# B&R Automation Studio project NAINV104C00R8L515F00 (part 7)

#### fHermesFormBoardArrived.st
```iecst
(* Hermes Form Board Arrived Table Data (Total Index Written In Table) *)
FUNCTION fHermesFormBoardArrived

	memset(ADR(pa_tyXMLTable) , 0 , SIZEOF(pa_tyXMLTable));
	iTotalIdxWrite	:= 0;

	fHermesGetTimestamp(ADR(sTimestamp) , tyDTStructure);

	pa_tyXMLTable[iTotalIdxWrite].sTitle	:= 'ST';
	pa_tyXMLTable[iTotalIdxWrite].sValue	:= 'Hermes';
	pa_tyXMLTable[iTotalIdxWrite].uiSize	:= LEN(pa_tyXMLTable[iTotalIdxWrite].sValue);

	iTotalIdxWrite	:= iTotalIdxWrite + 1;

	pa_tyXMLTable[iTotalIdxWrite].sTitle	:= 'AT';
	pa_tyXMLTable[iTotalIdxWrite].sValue	:= 'Timestamp';
	pa_tyXMLTable[iTotalIdxWrite].uiSize	:= LEN(pa_tyXMLTable[iTotalIdxWrite].sValue);

	iTotalIdxWrite	:= iTotalIdxWrite + 1;

	pa_tyXMLTable[iTotalIdxWrite].sTitle	:= 'AV';
	pa_tyXMLTable[iTotalIdxWrite].sValue	:= sTimestamp;
	pa_tyXMLTable[iTotalIdxWrite].uiSize	:= LEN(pa_tyXMLTable[iTotalIdxWrite].sValue);

	iTotalIdxWrite	:= iTotalIdxWrite + 1;

	pa_tyXMLTable[iTotalIdxWrite].sTitle	:= 'EN';
	pa_tyXMLTable[iTotalIdxWrite].sValue	:= '';
	pa_tyXMLTable[iTotalIdxWrite].uiSize	:= LEN(pa_tyXMLTable[iTotalIdxWrite].sValue);

	iTotalIdxWrite	:= iTotalIdxWrite + 1;

	pa_tyXMLTable[iTotalIdxWrite].sTitle	:= 'ST';
	pa_tyXMLTable[iTotalIdxWrite].sValue	:= 'BoardArrived';
	pa_tyXMLTable[iTotalIdxWrite].uiSize	:= LEN(pa_tyXMLTable[iTotalIdxWrite].sValue);

	iTotalIdxWrite	:= iTotalIdxWrite + 1;

	IF tyParameter.tyAvl.bMachineId = TRUE THEN
		pa_tyXMLTable[iTotalIdxWrite].sTitle	:= 'AT';
		pa_tyXMLTable[iTotalIdxWrite].sValue	:= 'MachineId';
		pa_tyXMLTable[iTotalIdxWrite].uiSize	:= LEN(pa_tyXMLTable[iTotalIdxWrite].sValue);

		iTotalIdxWrite	:= iTotalIdxWrite + 1;

		pa_tyXMLTable[iTotalIdxWrite].sTitle	:= 'AV';
		pa_tyXMLTable[iTotalIdxWrite].sValue	:= tyParameter.tyData.sMachineId;
		pa_tyXMLTable[iTotalIdxWrite].uiSize	:= LEN(pa_tyXMLTable[iTotalIdxWrite].sValue);

		iTotalIdxWrite	:= iTotalIdxWrite + 1;
	END_IF

	IF tyParameter.tyAvl.bUpstreamLaneId = TRUE THEN
		pa_tyXMLTable[iTotalIdxWrite].sTitle	:= 'AT';
		pa_tyXMLTable[iTotalIdxWrite].sValue	:= 'UpstreamLaneId';
		pa_tyXMLTable[iTotalIdxWrite].uiSize	:= LEN(pa_tyXMLTable[iTotalIdxWrite].sValue);

		iTotalIdxWrite	:= iTotalIdxWrite + 1;

		pa_tyXMLTable[iTotalIdxWrite].sTitle	:= 'AV';
		pa_tyXMLTable[iTotalIdxWrite].sValue	:= UDINT_TO_STRING(tyParameter.tyData.iUpstreamLaneId);
		pa_tyXMLTable[iTotalIdxWrite].uiSize	:= LEN(pa_tyXMLTable[iTotalIdxWrite].sValue);

		iTotalIdxWrite	:= iTotalIdxWrite + 1;
	END_IF

	IF tyParameter.tyAvl.bUpstreamInterfaceId = TRUE THEN
		pa_tyXMLTable[iTotalIdxWrite].sTitle	:= 'AT';
		pa_tyXMLTable[iTotalIdxWrite].sValue	:= 'UpstreamInterfaceId';
		pa_tyXMLTable[iTotalIdxWrite].uiSize	:= LEN(pa_tyXMLTable[iTotalIdxWrite].sValue);

		iTotalIdxWrite	:= iTotalIdxWrite + 1;

		pa_tyXMLTable[iTotalIdxWrite].sTitle	:= 'AV';
		pa_tyXMLTable[iTotalIdxWrite].sValue	:= tyParameter.tyData.sUpstreamInterfaceId;
		pa_tyXMLTable[iTotalIdxWrite].uiSize	:= LEN(pa_tyXMLTable[iTotalIdxWrite].sValue);

		iTotalIdxWrite	:= iTotalIdxWrite + 1;
	END_IF

	IF tyParameter.tyAvl.bMagazineId = TRUE THEN
		pa_tyXMLTable[iTotalIdxWrite].sTitle	:= 'AT';
		pa_tyXMLTable[iTotalIdxWrite].sValue	:= 'MagazineId';
		pa_tyXMLTable[iTotalIdxWrite].uiSize	:= LEN(pa_tyXMLTable[iTotalIdxWrite].sValue);

		iTotalIdxWrite	:= iTotalIdxWrite + 1;

		pa_tyXMLTable[iTotalIdxWrite].sTitle	:= 'AV';
		pa_tyXMLTable[iTotalIdxWrite].sValue	:= tyParameter.tyData.sMagazineId;
		pa_tyXMLTable[iTotalIdxWrite].uiSize	:= LEN(pa_tyXMLTable[iTotalIdxWrite].sValue);

		iTotalIdxWrite	:= iTotalIdxWrite + 1;
	END_IF

	IF tyParameter.tyAvl.bSlotId = TRUE THEN
		pa_tyXMLTable[iTotalIdxWrite].sTitle	:= 'AT';
		pa_tyXMLTable[iTotalIdxWrite].sValue	:= 'SlotId';
		pa_tyXMLTable[iTotalIdxWrite].uiSize	:= LEN(pa_tyXMLTable[iTotalIdxWrite].sValue);

		iTotalIdxWrite	:= iTotalIdxWrite + 1;

		pa_tyXMLTable[iTotalIdxWrite].sTitle	:= 'AV';
		pa_tyXMLTable[iTotalIdxWrite].sValue	:= UDINT_TO_STRING(tyParameter.tyData.iSlotId);
		pa_tyXMLTable[iTotalIdxWrite].uiSize	:= LEN(pa_tyXMLTable[iTotalIdxWrite].sValue);

		iTotalIdxWrite	:= iTotalIdxWrite + 1;
	END_IF

	IF tyParameter.tyAvl.bBoardTransfer = TRUE THEN
		pa_tyXMLTable[iTotalIdxWrite].sTitle	:= 'AT';
		pa_tyXMLTable[iTotalIdxWrite].sValue	:= 'BoardTransfer';
		pa_tyXMLTable[iTotalIdxWrite].uiSize	:= LEN(pa_tyXMLTable[iTotalIdxWrite].sValue);

		iTotalIdxWrite	:= iTotalIdxWrite + 1;

		pa_tyXMLTable[iTotalIdxWrite].sTitle	:= 'AV';
		pa_tyXMLTable[iTotalIdxWrite].sValue	:= DINT_TO_STRING(UDINT_TO_DINT(tyParameter.tyData.eBoadTransfer));
		pa_tyXMLTable[iTotalIdxWrite].uiSize	:= LEN(pa_tyXMLTable[iTotalIdxWrite].sValue);

		iTotalIdxWrite	:= iTotalIdxWrite + 1;
	END_IF

	IF tyParameter.tyAvl.bBoardId = TRUE THEN
		pa_tyXMLTable[iTotalIdxWrite].sTitle	:= 'AT';
		pa_tyXMLTable[iTotalIdxWrite].sValue	:= 'BoardId';
		pa_tyXMLTable[iTotalIdxWrite].uiSize	:= LEN(pa_tyXMLTable[iTotalIdxWrite].sValue);

		iTotalIdxWrite	:= iTotalIdxWrite + 1;

		pa_tyXMLTable[iTotalIdxWrite].sTitle	:= 'AV';
		pa_tyXMLTable[iTotalIdxWrite].sValue	:= tyParameter.tyData.sBoardId;
		pa_tyXMLTable[iTotalIdxWrite].uiSize	:= LEN(pa_tyXMLTable[iTotalIdxWrite].sValue);

		iTotalIdxWrite	:= iTotalIdxWrite + 1;
	END_IF

	IF tyParameter.tyAvl.bBoardIdCreatedBy = TRUE THEN
		pa_tyXMLTable[iTotalIdxWrite].sTitle	:= 'AT';
		pa_tyXMLTable[iTotalIdxWrite].sValue	:= 'BoardIdCreatedBy';
		pa_tyXMLTable[iTotalIdxWrite].uiSize	:= LEN(pa_tyXMLTable[iTotalIdxWrite].sValue);

		iTotalIdxWrite	:= iTotalIdxWrite + 1;

		pa_tyXMLTable[iTotalIdxWrite].sTitle	:= 'AV';
		pa_tyXMLTable[iTotalIdxWrite].sValue	:= tyParameter.tyData.sBoardIdCreatedBy;
		pa_tyXMLTable[iTotalIdxWrite].uiSize	:= LEN(pa_tyXMLTable[iTotalIdxWrite].sValue);

		iTotalIdxWrite	:= iTotalIdxWrite + 1;
	END_IF

	IF tyParameter.tyAvl.bFailedBoard = TRUE THEN
		pa_tyXMLTable[iTotalIdxWrite].sTitle	:= 'AT';
		pa_tyXMLTable[iTotalIdxWrite].sValue	:= 'FailedBoard';
		pa_tyXMLTable[iTotalIdxWrite].uiSize	:= LEN(pa_tyXMLTable[iTotalIdxWrite].sValue);

		iTotalIdxWrite	:= iTotalIdxWrite + 1;

		pa_tyXMLTable[iTotalIdxWrite].sTitle	:= 'AV';
		pa_tyXMLTable[iTotalIdxWrite].sValue	:= DINT_TO_STRING(UDINT_TO_DINT(tyParameter.tyData.eFailedBoard));
		pa_tyXMLTable[iTotalIdxWrite].uiSize	:= LEN(pa_tyXMLTable[iTotalIdxWrite].sValue);

		iTotalIdxWrite	:= iTotalIdxWrite + 1;
	END_IF

	IF tyParameter.tyAvl.bProductTypeId = TRUE THEN
		pa_tyXMLTable[iTotalIdxWrite].sTitle	:= 'AT';
		pa_tyXMLTable[iTotalIdxWrite].sValue	:= 'ProductTypeId';
		pa_tyXMLTable[iTotalIdxWrite].uiSize	:= LEN(pa_tyXMLTable[iTotalIdxWrite].sValue);

		iTotalIdxWrite	:= iTotalIdxWrite + 1;

		pa_tyXMLTable[iTotalIdxWrite].sTitle	:= 'AV';
		pa_tyXMLTable[iTotalIdxWrite].sValue	:= tyParameter.tyData.sProductTypeId;
		pa_tyXMLTable[iTotalIdxWrite].uiSize	:= LEN(pa_tyXMLTable[iTotalIdxWrite].sValue);

		iTotalIdxWrite	:= iTotalIdxWrite + 1;
	END_IF

	IF tyParameter.tyAvl.bFlippedBoard = TRUE THEN
		pa_tyXMLTable[iTotalIdxWrite].sTitle	:= 'AT';
		pa_tyXMLTable[iTotalIdxWrite].sValue	:= 'FlippedBoard';
		pa_tyXMLTable[iTotalIdxWrite].uiSize	:= LEN(pa_tyXMLTable[iTotalIdxWrite].sValue);

		iTotalIdxWrite	:= iTotalIdxWrite + 1;

		pa_tyXMLTable[iTotalIdxWrite].sTitle	:= 'AV';
		pa_tyXMLTable[iTotalIdxWrite].sValue	:= DINT_TO_STRING(UDINT_TO_DINT(tyParameter.tyData.eFlippedBoard));
		pa_tyXMLTable[iTotalIdxWrite].uiSize	:= LEN(pa_tyXMLTable[iTotalIdxWrite].sValue);

		iTotalIdxWrite	:= iTotalIdxWrite + 1;
	END_IF

	IF tyParameter.tyAvl.bTopBarcode = TRUE THEN
		pa_tyXMLTable[iTotalIdxWrite].sTitle	:= 'AT';
		pa_tyXMLTable[iTotalIdxWrite].sValue	:= 'TopBarcode';
		pa_tyXMLTable[iTotalIdxWrite].uiSize	:= LEN(pa_tyXMLTable[iTotalIdxWrite].sValue);

		iTotalIdxWrite	:= iTotalIdxWrite + 1;

		pa_tyXMLTable[iTotalIdxWrite].sTitle	:= 'AV';
		pa_tyXMLTable[iTotalIdxWrite].sValue	:= tyParameter.tyData.sTopBarcode;
		pa_tyXMLTable[iTotalIdxWrite].uiSize	:= LEN(pa_tyXMLTable[iTotalIdxWrite].sValue);

		iTotalIdxWrite	:= iTotalIdxWrite + 1;
	END_IF

	IF tyParameter.tyAvl.bBottomBarcode = TRUE THEN
		pa_tyXMLTable[iTotalIdxWrite].sTitle	:= 'AT';
		pa_tyXMLTable[iTotalIdxWrite].sValue	:= 'BottomBarcode';
		pa_tyXMLTable[iTotalIdxWrite].uiSize	:= LEN(pa_tyXMLTable[iTotalIdxWrite].sValue);

		iTotalIdxWrite	:= iTotalIdxWrite + 1;

		pa_tyXMLTable[iTotalIdxWrite].sTitle	:= 'AV';
		pa_tyXMLTable[iTotalIdxWrite].sValue	:= tyParameter.tyData.sBottomBarcode;
		pa_tyXMLTable[iTotalIdxWrite].uiSize	:= LEN(pa_tyXMLTable[iTotalIdxWrite].sValue);

		iTotalIdxWrite	:= iTotalIdxWrite + 1;
	END_IF

	IF tyParameter.tyAvl.bLength = TRUE THEN
		pa_tyXMLTable[iTotalIdxWrite].sTitle	:= 'AT';
		pa_tyXMLTable[iTotalIdxWrite].sValue	:= 'Length';
		pa_tyXMLTable[iTotalIdxWrite].uiSize	:= LEN(pa_tyXMLTable[iTotalIdxWrite].sValue);

		iTotalIdxWrite	:= iTotalIdxWrite + 1;

		pa_tyXMLTable[iTotalIdxWrite].sTitle	:= 'AV';
		pa_tyXMLTable[iTotalIdxWrite].sValue	:= REAL_TO_STRING(tyParameter.tyData.rLength);
		pa_tyXMLTable[iTotalIdxWrite].uiSize	:= LEN(pa_tyXMLTable[iTotalIdxWrite].sValue);

		iTotalIdxWrite	:= iTotalIdxWrite + 1;
	END_IF

	IF tyParameter.tyAvl.bWidth = TRUE THEN
		pa_tyXMLTable[iTotalIdxWrite].sTitle	:= 'AT';
		pa_tyXMLTable[iTotalIdxWrite].sValue	:= 'Width';
		pa_tyXMLTable[iTotalIdxWrite].uiSize	:= LEN(pa_tyXMLTable[iTotalIdxWrite].sValue);

		iTotalIdxWrite	:= iTotalIdxWrite + 1;

		pa_tyXMLTable[iTotalIdxWrite].sTitle	:= 'AV';
		pa_tyXMLTable[iTotalIdxWrite].sValue	:= REAL_TO_STRING(tyParameter.tyData.rWidth);
		pa_tyXMLTable[iTotalIdxWrite].uiSize	:= LEN(pa_tyXMLTable[iTotalIdxWrite].sValue);

		iTotalIdxWrite	:= iTotalIdxWrite + 1;
	END_IF

	IF tyParameter.tyAvl.bThickness = TRUE THEN
		pa_tyXMLTable[iTotalIdxWrite].sTitle	:= 'AT';
		pa_tyXMLTable[iTotalIdxWrite].sValue	:= 'Thickness';
		pa_tyXMLTable[iTotalIdxWrite].uiSize	:= LEN(pa_tyXMLTable[iTotalIdxWrite].sValue);

		iTotalIdxWrite	:= iTotalIdxWrite + 1;

		pa_tyXMLTable[iTotalIdxWrite].sTitle	:= 'AV';
		pa_tyXMLTable[iTotalIdxWrite].sValue	:= REAL_TO_STRING(tyParameter.tyData.rThickness);
		pa_tyXMLTable[iTotalIdxWrite].uiSize	:= LEN(pa_tyXMLTable[iTotalIdxWrite].sValue);

		iTotalIdxWrite	:= iTotalIdxWrite + 1;
	END_IF

	IF tyParameter.tyAvl.bConveyorSpeed = TRUE THEN
		pa_tyXMLTable[iTotalIdxWrite].sTitle	:= 'AT';
		pa_tyXMLTable[iTotalIdxWrite].sValue	:= 'ConveyorSpeed';
		pa_tyXMLTable[iTotalIdxWrite].uiSize	:= LEN(pa_tyXMLTable[iTotalIdxWrite].sValue);

		iTotalIdxWrite	:= iTotalIdxWrite + 1;

		pa_tyXMLTable[iTotalIdxWrite].sTitle	:= 'AV';
		pa_tyXMLTable[iTotalIdxWrite].sValue	:= REAL_TO_STRING(tyParameter.tyData.rConveyorSpeed);
		pa_tyXMLTable[iTotalIdxWrite].uiSize	:= LEN(pa_tyXMLTable[iTotalIdxWrite].sValue);

		iTotalIdxWrite	:= iTotalIdxWrite + 1;
	END_IF

	IF tyParameter.tyAvl.bTopClearanceHeight = TRUE THEN
		pa_tyXMLTable[iTotalIdxWrite].sTitle	:= 'AT';
		pa_tyXMLTable[iTotalIdxWrite].sValue	:= 'TopClearanceHeight';
		pa_tyXMLTable[iTotalIdxWrite].uiSize	:= LEN(pa_tyXMLTable[iTotalIdxWrite].sValue);

		iTotalIdxWrite	:= iTotalIdxWrite + 1;

		pa_tyXMLTable[iTotalIdxWrite].sTitle	:= 'AV';
		pa_tyXMLTable[iTotalIdxWrite].sValue	:= REAL_TO_STRING(tyParameter.tyData.rTopClearanceHeight);
		pa_tyXMLTable[iTotalIdxWrite].uiSize	:= LEN(pa_tyXMLTable[iTotalIdxWrite].sValue);

		iTotalIdxWrite	:= iTotalIdxWrite + 1;
	END_IF

	IF tyParameter.tyAvl.bBottomClearanceHeight = TRUE THEN
		pa_tyXMLTable[iTotalIdxWrite].sTitle	:= 'AT';
		pa_tyXMLTable[iTotalIdxWrite].sValue	:= 'BottomClearanceHeight';
		pa_tyXMLTable[iTotalIdxWrite].uiSize	:= LEN(pa_tyXMLTable[iTotalIdxWrite].sValue);

		iTotalIdxWrite	:= iTotalIdxWrite + 1;

		pa_tyXMLTable[iTotalIdxWrite].sTitle	:= 'AV';
		pa_tyXMLTable[iTotalIdxWrite].sValue	:= REAL_TO_STRING(tyParameter.tyData.rBottomClearanceHeight);
		pa_tyXMLTable[iTotalIdxWrite].uiSize	:= LEN(pa_tyXMLTable[iTotalIdxWrite].sValue);

		iTotalIdxWrite	:= iTotalIdxWrite + 1;
	END_IF

	IF tyParameter.tyAvl.bWeight = TRUE THEN
		pa_tyXMLTable[iTotalIdxWrite].sTitle	:= 'AT';
		pa_tyXMLTable[iTotalIdxWrite].sValue	:= 'Weight';
		pa_tyXMLTable[iTotalIdxWrite].uiSize	:= LEN(pa_tyXMLTable[iTotalIdxWrite].sValue);

		iTotalIdxWrite	:= iTotalIdxWrite + 1;

		pa_tyXMLTable[iTotalIdxWrite].sTitle	:= 'AV';
		pa_tyXMLTable[iTotalIdxWrite].sValue	:= REAL_TO_STRING(tyParameter.tyData.rWeight);
		pa_tyXMLTable[iTotalIdxWrite].uiSize	:= LEN(pa_tyXMLTable[iTotalIdxWrite].sValue);

		iTotalIdxWrite	:= iTotalIdxWrite + 1;
	END_IF

	IF tyParameter.tyAvl.bWorkOrderId = TRUE THEN
		pa_tyXMLTable[iTotalIdxWrite].sTitle	:= 'AT';
		pa_tyXMLTable[iTotalIdxWrite].sValue	:= 'WorkOrderId';
		pa_tyXMLTable[iTotalIdxWrite].uiSize	:= LEN(pa_tyXMLTable[iTotalIdxWrite].sValue);

		iTotalIdxWrite	:= iTotalIdxWrite + 1;

		pa_tyXMLTable[iTotalIdxWrite].sTitle	:= 'AV';
		pa_tyXMLTable[iTotalIdxWrite].sValue	:= tyParameter.tyData.sWorkOrdedId;
		pa_tyXMLTable[iTotalIdxWrite].uiSize	:= LEN(pa_tyXMLTable[iTotalIdxWrite].sValue);

		iTotalIdxWrite	:= iTotalIdxWrite + 1;
	END_IF

	IF tyParameter.tyAvl.bBatchId = TRUE THEN
		pa_tyXMLTable[iTotalIdxWrite].sTitle	:= 'AT';
		pa_tyXMLTable[iTotalIdxWrite].sValue	:= 'BatchId';
		pa_tyXMLTable[iTotalIdxWrite].uiSize	:= LEN(pa_tyXMLTable[iTotalIdxWrite].sValue);

		iTotalIdxWrite	:= iTotalIdxWrite + 1;

		pa_tyXMLTable[iTotalIdxWrite].sTitle	:= 'AV';
		pa_tyXMLTable[iTotalIdxWrite].sValue	:= tyParameter.tyData.sBatchId;
		pa_tyXMLTable[iTotalIdxWrite].uiSize	:= LEN(pa_tyXMLTable[iTotalIdxWrite].sValue);

		iTotalIdxWrite	:= iTotalIdxWrite + 1;
	END_IF

	IF tyParameter.tyAvl.bRoute = TRUE THEN
		pa_tyXMLTable[iTotalIdxWrite].sTitle	:= 'AT';
		pa_tyXMLTable[iTotalIdxWrite].sValue	:= 'Route';
		pa_tyXMLTable[iTotalIdxWrite].uiSize	:= LEN(pa_tyXMLTable[iTotalIdxWrite].sValue);

		iTotalIdxWrite	:= iTotalIdxWrite + 1;

		pa_tyXMLTable[iTotalIdxWrite].sTitle	:= 'AV';
		pa_tyXMLTable[iTotalIdxWrite].sValue	:= INT_TO_STRING(tyParameter.tyData.iRoute);
		pa_tyXMLTable[iTotalIdxWrite].uiSize	:= LEN(pa_tyXMLTable[iTotalIdxWrite].sValue);

		iTotalIdxWrite	:= iTotalIdxWrite + 1;
	END_IF

	IF tyParameter.tyAvl.bAction = TRUE THEN
		pa_tyXMLTable[iTotalIdxWrite].sTitle	:= 'AT';
		pa_tyXMLTable[iTotalIdxWrite].sValue	:= 'Action';
		pa_tyXMLTable[iTotalIdxWrite].uiSize	:= LEN(pa_tyXMLTable[iTotalIdxWrite].sValue);

		iTotalIdxWrite	:= iTotalIdxWrite + 1;

		pa_tyXMLTable[iTotalIdxWrite].sTitle	:= 'AV';
		pa_tyXMLTable[iTotalIdxWrite].sValue	:= INT_TO_STRING(tyParameter.tyData.iAction);
		pa_tyXMLTable[iTotalIdxWrite].uiSize	:= LEN(pa_tyXMLTable[iTotalIdxWrite].sValue);

		iTotalIdxWrite	:= iTotalIdxWrite + 1;
	END_IF

	pa_tyXMLTable[iTotalIdxWrite].sTitle	:= 'ES';
	pa_tyXMLTable[iTotalIdxWrite].sValue	:= '';
	pa_tyXMLTable[iTotalIdxWrite].uiSize	:= LEN(pa_tyXMLTable[iTotalIdxWrite].sValue);

	iTotalIdxWrite	:= iTotalIdxWrite + 1;

	pa_tyXMLTable[iTotalIdxWrite].sTitle	:= 'ET';
	pa_tyXMLTable[iTotalIdxWrite].sValue	:= 'Hermes';
	pa_tyXMLTable[iTotalIdxWrite].uiSize	:= LEN(pa_tyXMLTable[iTotalIdxWrite].sValue);

	iTotalIdxWrite	:= iTotalIdxWrite + 1;

	pa_tyXMLTable[iTotalIdxWrite].sTitle	:= 'EN';
	pa_tyXMLTable[iTotalIdxWrite].sValue	:= '';
	pa_tyXMLTable[iTotalIdxWrite].uiSize	:= LEN(pa_tyXMLTable[iTotalIdxWrite].sValue);

	iTotalIdxWrite	:= iTotalIdxWrite + 1;

	iTotalIdxWrite	:= fHermesFormBoardArrived;

END_FUNCTION
```

#### fHermesFormBoardDeparted.st
```iecst
(* Hermes Form Board Departed Table Data (Total Index Written In Table) *)
FUNCTION fHermesFormBoardDeparted

	memset(ADR(pa_tyXMLTable) , 0 , SIZEOF(pa_tyXMLTable));
	iTotalIdxWrite	:= 0;

	fHermesGetTimestamp(ADR(sTimestamp) , tyDTStructure);

	pa_tyXMLTable[iTotalIdxWrite].sTitle	:= 'ST';
	pa_tyXMLTable[iTotalIdxWrite].sValue	:= 'Hermes';
	pa_tyXMLTable[iTotalIdxWrite].uiSize	:= LEN(pa_tyXMLTable[iTotalIdxWrite].sValue);

	iTotalIdxWrite	:= iTotalIdxWrite + 1;

	pa_tyXMLTable[iTotalIdxWrite].sTitle	:= 'AT';
	pa_tyXMLTable[iTotalIdxWrite].sValue	:= 'Timestamp';
	pa_tyXMLTable[iTotalIdxWrite].uiSize	:= LEN(pa_tyXMLTable[iTotalIdxWrite].sValue);

	iTotalIdxWrite	:= iTotalIdxWrite + 1;

	pa_tyXMLTable[iTotalIdxWrite].sTitle	:= 'AV';
	pa_tyXMLTable[iTotalIdxWrite].sValue	:= sTimestamp;
	pa_tyXMLTable[iTotalIdxWrite].uiSize	:= LEN(pa_tyXMLTable[iTotalIdxWrite].sValue);

	iTotalIdxWrite	:= iTotalIdxWrite + 1;

	pa_tyXMLTable[iTotalIdxWrite].sTitle	:= 'EN';
	pa_tyXMLTable[iTotalIdxWrite].sValue	:= '';
	pa_tyXMLTable[iTotalIdxWrite].uiSize	:= LEN(pa_tyXMLTable[iTotalIdxWrite].sValue);

	iTotalIdxWrite	:= iTotalIdxWrite + 1;

	pa_tyXMLTable[iTotalIdxWrite].sTitle	:= 'ST';
	pa_tyXMLTable[iTotalIdxWrite].sValue	:= 'BoardDeparted';
	pa_tyXMLTable[iTotalIdxWrite].uiSize	:= LEN(pa_tyXMLTable[iTotalIdxWrite].sValue);

	iTotalIdxWrite	:= iTotalIdxWrite + 1;

	IF tyParameter.tyAvl.bMachineId = TRUE THEN
		pa_tyXMLTable[iTotalIdxWrite].sTitle	:= 'AT';
		pa_tyXMLTable[iTotalIdxWrite].sValue	:= 'MachineId';
		pa_tyXMLTable[iTotalIdxWrite].uiSize	:= LEN(pa_tyXMLTable[iTotalIdxWrite].sValue);

		iTotalIdxWrite	:= iTotalIdxWrite + 1;

		pa_tyXMLTable[iTotalIdxWrite].sTitle	:= 'AV';
		pa_tyXMLTable[iTotalIdxWrite].sValue	:= tyParameter.tyData.sMachineId;
		pa_tyXMLTable[iTotalIdxWrite].uiSize	:= LEN(pa_tyXMLTable[iTotalIdxWrite].sValue);

		iTotalIdxWrite	:= iTotalIdxWrite + 1;
	END_IF

	IF tyParameter.tyAvl.bDownstreamLaneId = TRUE THEN
		pa_tyXMLTable[iTotalIdxWrite].sTitle	:= 'AT';
		pa_tyXMLTable[iTotalIdxWrite].sValue	:= 'DownstreamLaneId';
		pa_tyXMLTable[iTotalIdxWrite].uiSize	:= LEN(pa_tyXMLTable[iTotalIdxWrite].sValue);

		iTotalIdxWrite	:= iTotalIdxWrite + 1;

		pa_tyXMLTable[iTotalIdxWrite].sTitle	:= 'AV';
		pa_tyXMLTable[iTotalIdxWrite].sValue	:= UDINT_TO_STRING(tyParameter.tyData.iDownstreamLaneId);
		pa_tyXMLTable[iTotalIdxWrite].uiSize	:= LEN(pa_tyXMLTable[iTotalIdxWrite].sValue);

		iTotalIdxWrite	:= iTotalIdxWrite + 1;
	END_IF

	IF tyParameter.tyAvl.bDownstreamInterfaceId = TRUE THEN
		pa_tyXMLTable[iTotalIdxWrite].sTitle	:= 'AT';
		pa_tyXMLTable[iTotalIdxWrite].sValue	:= 'DownstreamInterfaceId';
		pa_tyXMLTable[iTotalIdxWrite].uiSize	:= LEN(pa_tyXMLTable[iTotalIdxWrite].sValue);

		iTotalIdxWrite	:= iTotalIdxWrite + 1;

		pa_tyXMLTable[iTotalIdxWrite].sTitle	:= 'AV';
		pa_tyXMLTable[iTotalIdxWrite].sValue	:= tyParameter.tyData.sDownstreamInterfaceId;
		pa_tyXMLTable[iTotalIdxWrite].uiSize	:= LEN(pa_tyXMLTable[iTotalIdxWrite].sValue);

		iTotalIdxWrite	:= iTotalIdxWrite + 1;
	END_IF

	IF tyParameter.tyAvl.bMagazineId = TRUE THEN
		pa_tyXMLTable[iTotalIdxWrite].sTitle	:= 'AT';
		pa_tyXMLTable[iTotalIdxWrite].sValue	:= 'MagazineId';
		pa_tyXMLTable[iTotalIdxWrite].uiSize	:= LEN(pa_tyXMLTable[iTotalIdxWrite].sValue);

		iTotalIdxWrite	:= iTotalIdxWrite + 1;

		pa_tyXMLTable[iTotalIdxWrite].sTitle	:= 'AV';
		pa_tyXMLTable[iTotalIdxWrite].sValue	:= tyParameter.tyData.sMagazineId;
		pa_tyXMLTable[iTotalIdxWrite].uiSize	:= LEN(pa_tyXMLTable[iTotalIdxWrite].sValue);

		iTotalIdxWrite	:= iTotalIdxWrite + 1;
	END_IF

	IF tyParameter.tyAvl.bSlotId = TRUE THEN
		pa_tyXMLTable[iTotalIdxWrite].sTitle	:= 'AT';
		pa_tyXMLTable[iTotalIdxWrite].sValue	:= 'SlotId';
		pa_tyXMLTable[iTotalIdxWrite].uiSize	:= LEN(pa_tyXMLTable[iTotalIdxWrite].sValue);

		iTotalIdxWrite	:= iTotalIdxWrite + 1;

		pa_tyXMLTable[iTotalIdxWrite].sTitle	:= 'AV';
		pa_tyXMLTable[iTotalIdxWrite].sValue	:= UDINT_TO_STRING(tyParameter.tyData.iSlotId);
		pa_tyXMLTable[iTotalIdxWrite].uiSize	:= LEN(pa_tyXMLTable[iTotalIdxWrite].sValue);

		iTotalIdxWrite	:= iTotalIdxWrite + 1;
	END_IF

	IF tyParameter.tyAvl.bBoardTransfer = TRUE THEN
		pa_tyXMLTable[iTotalIdxWrite].sTitle	:= 'AT';
		pa_tyXMLTable[iTotalIdxWrite].sValue	:= 'BoardTransfer';
		pa_tyXMLTable[iTotalIdxWrite].uiSize	:= LEN(pa_tyXMLTable[iTotalIdxWrite].sValue);

		iTotalIdxWrite	:= iTotalIdxWrite + 1;

		pa_tyXMLTable[iTotalIdxWrite].sTitle	:= 'AV';
		pa_tyXMLTable[iTotalIdxWrite].sValue	:= DINT_TO_STRING(UDINT_TO_DINT(tyParameter.tyData.eBoadTransfer));
		pa_tyXMLTable[iTotalIdxWrite].uiSize	:= LEN(pa_tyXMLTable[iTotalIdxWrite].sValue);

		iTotalIdxWrite	:= iTotalIdxWrite + 1;
	END_IF

	IF tyParameter.tyAvl.bBoardId = TRUE THEN
		pa_tyXMLTable[iTotalIdxWrite].sTitle	:= 'AT';
		pa_tyXMLTable[iTotalIdxWrite].sValue	:= 'BoardId';
		pa_tyXMLTable[iTotalIdxWrite].uiSize	:= LEN(pa_tyXMLTable[iTotalIdxWrite].sValue);

		iTotalIdxWrite	:= iTotalIdxWrite + 1;

		pa_tyXMLTable[iTotalIdxWrite].sTitle	:= 'AV';
		pa_tyXMLTable[iTotalIdxWrite].sValue	:= tyParameter.tyData.sBoardId;
		pa_tyXMLTable[iTotalIdxWrite].uiSize	:= LEN(pa_tyXMLTable[iTotalIdxWrite].sValue);

		iTotalIdxWrite	:= iTotalIdxWrite + 1;
	END_IF

	IF tyParameter.tyAvl.bBoardIdCreatedBy = TRUE THEN
		pa_tyXMLTable[iTotalIdxWrite].sTitle	:= 'AT';
		pa_tyXMLTable[iTotalIdxWrite].sValue	:= 'BoardIdCreatedBy';
		pa_tyXMLTable[iTotalIdxWrite].uiSize	:= LEN(pa_tyXMLTable[iTotalIdxWrite].sValue);

		iTotalIdxWrite	:= iTotalIdxWrite + 1;

		pa_tyXMLTable[iTotalIdxWrite].sTitle	:= 'AV';
		pa_tyXMLTable[iTotalIdxWrite].sValue	:= tyParameter.tyData.sBoardIdCreatedBy;
		pa_tyXMLTable[iTotalIdxWrite].uiSize	:= LEN(pa_tyXMLTable[iTotalIdxWrite].sValue);

		iTotalIdxWrite	:= iTotalIdxWrite + 1;
	END_IF

	IF tyParameter.tyAvl.bFailedBoard = TRUE THEN
		pa_tyXMLTable[iTotalIdxWrite].sTitle	:= 'AT';
		pa_tyXMLTable[iTotalIdxWrite].sValue	:= 'FailedBoard';
		pa_tyXMLTable[iTotalIdxWrite].uiSize	:= LEN(pa_tyXMLTable[iTotalIdxWrite].sValue);

		iTotalIdxWrite	:= iTotalIdxWrite + 1;

		pa_tyXMLTable[iTotalIdxWrite].sTitle	:= 'AV';
		pa_tyXMLTable[iTotalIdxWrite].sValue	:= DINT_TO_STRING(UDINT_TO_DINT(tyParameter.tyData.eFailedBoard));
		pa_tyXMLTable[iTotalIdxWrite].uiSize	:= LEN(pa_tyXMLTable[iTotalIdxWrite].sValue);

		iTotalIdxWrite	:= iTotalIdxWrite + 1;
	END_IF

	IF tyParameter.tyAvl.bProductTypeId = TRUE THEN
		pa_tyXMLTable[iTotalIdxWrite].sTitle	:= 'AT';
		pa_tyXMLTable[iTotalIdxWrite].sValue	:= 'ProductTypeId';
		pa_tyXMLTable[iTotalIdxWrite].uiSize	:= LEN(pa_tyXMLTable[iTotalIdxWrite].sValue);

		iTotalIdxWrite	:= iTotalIdxWrite + 1;

		pa_tyXMLTable[iTotalIdxWrite].sTitle	:= 'AV';
		pa_tyXMLTable[iTotalIdxWrite].sValue	:= tyParameter.tyData.sProductTypeId;
		pa_tyXMLTable[iTotalIdxWrite].uiSize	:= LEN(pa_tyXMLTable[iTotalIdxWrite].sValue);

		iTotalIdxWrite	:= iTotalIdxWrite + 1;
	END_IF

	IF tyParameter.tyAvl.bFlippedBoard = TRUE THEN
		pa_tyXMLTable[iTotalIdxWrite].sTitle	:= 'AT';
		pa_tyXMLTable[iTotalIdxWrite].sValue	:= 'FlippedBoard';
		pa_tyXMLTable[iTotalIdxWrite].uiSize	:= LEN(pa_tyXMLTable[iTotalIdxWrite].sValue);

		iTotalIdxWrite	:= iTotalIdxWrite + 1;

		pa_tyXMLTable[iTotalIdxWrite].sTitle	:= 'AV';
		pa_tyXMLTable[iTotalIdxWrite].sValue	:= DINT_TO_STRING(UDINT_TO_DINT(tyParameter.tyData.eFlippedBoard));
		pa_tyXMLTable[iTotalIdxWrite].uiSize	:= LEN(pa_tyXMLTable[iTotalIdxWrite].sValue);

		iTotalIdxWrite	:= iTotalIdxWrite + 1;
	END_IF

	IF tyParameter.tyAvl.bTopBarcode = TRUE THEN
		pa_tyXMLTable[iTotalIdxWrite].sTitle	:= 'AT';
		pa_tyXMLTable[iTotalIdxWrite].sValue	:= 'TopBarcode';
		pa_tyXMLTable[iTotalIdxWrite].uiSize	:= LEN(pa_tyXMLTable[iTotalIdxWrite].sValue);

		iTotalIdxWrite	:= iTotalIdxWrite + 1;

		pa_tyXMLTable[iTotalIdxWrite].sTitle	:= 'AV';
		pa_tyXMLTable[iTotalIdxWrite].sValue	:= tyParameter.tyData.sTopBarcode;
		pa_tyXMLTable[iTotalIdxWrite].uiSize	:= LEN(pa_tyXMLTable[iTotalIdxWrite].sValue);

		iTotalIdxWrite	:= iTotalIdxWrite + 1;
	END_IF

	IF tyParameter.tyAvl.bBottomBarcode = TRUE THEN
		pa_tyXMLTable[iTotalIdxWrite].sTitle	:= 'AT';
		pa_tyXMLTable[iTotalIdxWrite].sValue	:= 'BottomBarcode';
		pa_tyXMLTable[iTotalIdxWrite].uiSize	:= LEN(pa_tyXMLTable[iTotalIdxWrite].sValue);

		iTotalIdxWrite	:= iTotalIdxWrite + 1;

		pa_tyXMLTable[iTotalIdxWrite].sTitle	:= 'AV';
		pa_tyXMLTable[iTotalIdxWrite].sValue	:= tyParameter.tyData.sBottomBarcode;
		pa_tyXMLTable[iTotalIdxWrite].uiSize	:= LEN(pa_tyXMLTable[iTotalIdxWrite].sValue);

		iTotalIdxWrite	:= iTotalIdxWrite + 1;
	END_IF

	IF tyParameter.tyAvl.bLength = TRUE THEN
		pa_tyXMLTable[iTotalIdxWrite].sTitle	:= 'AT';
		pa_tyXMLTable[iTotalIdxWrite].sValue	:= 'Length';
		pa_tyXMLTable[iTotalIdxWrite].uiSize	:= LEN(pa_tyXMLTable[iTotalIdxWrite].sValue);

		iTotalIdxWrite	:= iTotalIdxWrite + 1;

		pa_tyXMLTable[iTotalIdxWrite].sTitle	:= 'AV';
		pa_tyXMLTable[iTotalIdxWrite].sValue	:= REAL_TO_STRING(tyParameter.tyData.rLength);
		pa_tyXMLTable[iTotalIdxWrite].uiSize	:= LEN(pa_tyXMLTable[iTotalIdxWrite].sValue);

		iTotalIdxWrite	:= iTotalIdxWrite + 1;
	END_IF

	IF tyParameter.tyAvl.bWidth = TRUE THEN
		pa_tyXMLTable[iTotalIdxWrite].sTitle	:= 'AT';
		pa_tyXMLTable[iTotalIdxWrite].sValue	:= 'Width';
		pa_tyXMLTable[iTotalIdxWrite].uiSize	:= LEN(pa_tyXMLTable[iTotalIdxWrite].sValue);

		iTotalIdxWrite	:= iTotalIdxWrite + 1;

		pa_tyXMLTable[iTotalIdxWrite].sTitle	:= 'AV';
		pa_tyXMLTable[iTotalIdxWrite].sValue	:= REAL_TO_STRING(tyParameter.tyData.rWidth);
		pa_tyXMLTable[iTotalIdxWrite].uiSize	:= LEN(pa_tyXMLTable[iTotalIdxWrite].sValue);

		iTotalIdxWrite	:= iTotalIdxWrite + 1;
	END_IF

	IF tyParameter.tyAvl.bThickness = TRUE THEN
		pa_tyXMLTable[iTotalIdxWrite].sTitle	:= 'AT';
		pa_tyXMLTable[iTotalIdxWrite].sValue	:= 'Thickness';
		pa_tyXMLTable[iTotalIdxWrite].uiSize	:= LEN(pa_tyXMLTable[iTotalIdxWrite].sValue);

		iTotalIdxWrite	:= iTotalIdxWrite + 1;

		pa_tyXMLTable[iTotalIdxWrite].sTitle	:= 'AV';
		pa_tyXMLTable[iTotalIdxWrite].sValue	:= REAL_TO_STRING(tyParameter.tyData.rThickness);
		pa_tyXMLTable[iTotalIdxWrite].uiSize	:= LEN(pa_tyXMLTable[iTotalIdxWrite].sValue);

		iTotalIdxWrite	:= iTotalIdxWrite + 1;
	END_IF

	IF tyParameter.tyAvl.bConveyorSpeed = TRUE THEN
		pa_tyXMLTable[iTotalIdxWrite].sTitle	:= 'AT';
		pa_tyXMLTable[iTotalIdxWrite].sValue	:= 'ConveyorSpeed';
		pa_tyXMLTable[iTotalIdxWrite].uiSize	:= LEN(pa_tyXMLTable[iTotalIdxWrite].sValue);

		iTotalIdxWrite	:= iTotalIdxWrite + 1;

		pa_tyXMLTable[iTotalIdxWrite].sTitle	:= 'AV';
		pa_tyXMLTable[iTotalIdxWrite].sValue	:= REAL_TO_STRING(tyParameter.tyData.rConveyorSpeed);
		pa_tyXMLTable[iTotalIdxWrite].uiSize	:= LEN(pa_tyXMLTable[iTotalIdxWrite].sValue);

		iTotalIdxWrite	:= iTotalIdxWrite + 1;
	END_IF

	IF tyParameter.tyAvl.bTopClearanceHeight = TRUE THEN
		pa_tyXMLTable[iTotalIdxWrite].sTitle	:= 'AT';
		pa_tyXMLTable[iTotalIdxWrite].sValue	:= 'TopClearanceHeight';
		pa_tyXMLTable[iTotalIdxWrite].uiSize	:= LEN(pa_tyXMLTable[iTotalIdxWrite].sValue);

		iTotalIdxWrite	:= iTotalIdxWrite + 1;

		pa_tyXMLTable[iTotalIdxWrite].sTitle	:= 'AV';
		pa_tyXMLTable[iTotalIdxWrite].sValue	:= REAL_TO_STRING(tyParameter.tyData.rTopClearanceHeight);
		pa_tyXMLTable[iTotalIdxWrite].uiSize	:= LEN(pa_tyXMLTable[iTotalIdxWrite].sValue);

		iTotalIdxWrite	:= iTotalIdxWrite + 1;
	END_IF

	IF tyParameter.tyAvl.bBottomClearanceHeight = TRUE THEN
		pa_tyXMLTable[iTotalIdxWrite].sTitle	:= 'AT';
		pa_tyXMLTable[iTotalIdxWrite].sValue	:= 'BottomClearanceHeight';
		pa_tyXMLTable[iTotalIdxWrite].uiSize	:= LEN(pa_tyXMLTable[iTotalIdxWrite].sValue);

		iTotalIdxWrite	:= iTotalIdxWrite + 1;

		pa_tyXMLTable[iTotalIdxWrite].sTitle	:= 'AV';
		pa_tyXMLTable[iTotalIdxWrite].sValue	:= REAL_TO_STRING(tyParameter.tyData.rBottomClearanceHeight);
		pa_tyXMLTable[iTotalIdxWrite].uiSize	:= LEN(pa_tyXMLTable[iTotalIdxWrite].sValue);

		iTotalIdxWrite	:= iTotalIdxWrite + 1;
	END_IF

	IF tyParameter.tyAvl.bWeight = TRUE THEN
		pa_tyXMLTable[iTotalIdxWrite].sTitle	:= 'AT';
		pa_tyXMLTable[iTotalIdxWrite].sValue	:= 'Weight';
		pa_tyXMLTable[iTotalIdxWrite].uiSize	:= LEN(pa_tyXMLTable[iTotalIdxWrite].sValue);

		iTotalIdxWrite	:= iTotalIdxWrite + 1;

		pa_tyXMLTable[iTotalIdxWrite].sTitle	:= 'AV';
		pa_tyXMLTable[iTotalIdxWrite].sValue	:= REAL_TO_STRING(tyParameter.tyData.rWeight);
		pa_tyXMLTable[iTotalIdxWrite].uiSize	:= LEN(pa_tyXMLTable[iTotalIdxWrite].sValue);

		iTotalIdxWrite	:= iTotalIdxWrite + 1;
	END_IF

	IF tyParameter.tyAvl.bWorkOrderId = TRUE THEN
		pa_tyXMLTable[iTotalIdxWrite].sTitle	:= 'AT';
		pa_tyXMLTable[iTotalIdxWrite].sValue	:= 'WorkOrderId';
		pa_tyXMLTable[iTotalIdxWrite].uiSize	:= LEN(pa_tyXMLTable[iTotalIdxWrite].sValue);

		iTotalIdxWrite	:= iTotalIdxWrite + 1;

		pa_tyXMLTable[iTotalIdxWrite].sTitle	:= 'AV';
		pa_tyXMLTable[iTotalIdxWrite].sValue	:= tyParameter.tyData.sWorkOrdedId;
		pa_tyXMLTable[iTotalIdxWrite].uiSize	:= LEN(pa_tyXMLTable[iTotalIdxWrite].sValue);

		iTotalIdxWrite	:= iTotalIdxWrite + 1;
	END_IF

	IF tyParameter.tyAvl.bBatchId = TRUE THEN
		pa_tyXMLTable[iTotalIdxWrite].sTitle	:= 'AT';
		pa_tyXMLTable[iTotalIdxWrite].sValue	:= 'BatchId';
		pa_tyXMLTable[iTotalIdxWrite].uiSize	:= LEN(pa_tyXMLTable[iTotalIdxWrite].sValue);

		iTotalIdxWrite	:= iTotalIdxWrite + 1;

		pa_tyXMLTable[iTotalIdxWrite].sTitle	:= 'AV';
		pa_tyXMLTable[iTotalIdxWrite].sValue	:= tyParameter.tyData.sBatchId;
		pa_tyXMLTable[iTotalIdxWrite].uiSize	:= LEN(pa_tyXMLTable[iTotalIdxWrite].sValue);

		iTotalIdxWrite	:= iTotalIdxWrite + 1;
	END_IF

	pa_tyXMLTable[iTotalIdxWrite].sTitle	:= 'ES';
	pa_tyXMLTable[iTotalIdxWrite].sValue	:= '';
	pa_tyXMLTable[iTotalIdxWrite].uiSize	:= LEN(pa_tyXMLTable[iTotalIdxWrite].sValue);

	iTotalIdxWrite	:= iTotalIdxWrite + 1;

	pa_tyXMLTable[iTotalIdxWrite].sTitle	:= 'ET';
	pa_tyXMLTable[iTotalIdxWrite].sValue	:= 'Hermes';
	pa_tyXMLTable[iTotalIdxWrite].uiSize	:= LEN(pa_tyXMLTable[iTotalIdxWrite].sValue);

	iTotalIdxWrite	:= iTotalIdxWrite + 1;

	pa_tyXMLTable[iTotalIdxWrite].sTitle	:= 'EN';
	pa_tyXMLTable[iTotalIdxWrite].sValue	:= '';
	pa_tyXMLTable[iTotalIdxWrite].uiSize	:= LEN(pa_tyXMLTable[iTotalIdxWrite].sValue);

	iTotalIdxWrite	:= iTotalIdxWrite + 1;

	iTotalIdxWrite	:= fHermesFormBoardDeparted;

END_FUNCTION
```

#### fHermesFormQueryWorkOrderInfo.st
```iecst
(* Hermes Form Query WorkOrder Info Table Data (Total Index Written In Table) *)
FUNCTION fHermesFormQueryWorkOrderInfo

	memset(ADR(pa_tyXMLTable) , 0 , SIZEOF(pa_tyXMLTable));
	iTotalIdxWrite	:= 0;

	fHermesGetTimestamp(ADR(sTimestamp) , tyDTStructure);

	pa_tyXMLTable[iTotalIdxWrite].sTitle	:= 'ST';
	pa_tyXMLTable[iTotalIdxWrite].sValue	:= 'Hermes';
	pa_tyXMLTable[iTotalIdxWrite].uiSize	:= LEN(pa_tyXMLTable[iTotalIdxWrite].sValue);

	iTotalIdxWrite	:= iTotalIdxWrite + 1;

	pa_tyXMLTable[iTotalIdxWrite].sTitle	:= 'AT';
	pa_tyXMLTable[iTotalIdxWrite].sValue	:= 'Timestamp';
	pa_tyXMLTable[iTotalIdxWrite].uiSize	:= LEN(pa_tyXMLTable[iTotalIdxWrite].sValue);

	iTotalIdxWrite	:= iTotalIdxWrite + 1;

	pa_tyXMLTable[iTotalIdxWrite].sTitle	:= 'AV';
	pa_tyXMLTable[iTotalIdxWrite].sValue	:= sTimestamp;
	pa_tyXMLTable[iTotalIdxWrite].uiSize	:= LEN(pa_tyXMLTable[iTotalIdxWrite].sValue);

	iTotalIdxWrite	:= iTotalIdxWrite + 1;

	pa_tyXMLTable[iTotalIdxWrite].sTitle	:= 'EN';
	pa_tyXMLTable[iTotalIdxWrite].sValue	:= '';
	pa_tyXMLTable[iTotalIdxWrite].uiSize	:= LEN(pa_tyXMLTable[iTotalIdxWrite].sValue);

	iTotalIdxWrite	:= iTotalIdxWrite + 1;

	pa_tyXMLTable[iTotalIdxWrite].sTitle	:= 'ST';
	pa_tyXMLTable[iTotalIdxWrite].sValue	:= 'QueryWorkOrderInfo';
	pa_tyXMLTable[iTotalIdxWrite].uiSize	:= LEN(pa_tyXMLTable[iTotalIdxWrite].sValue);

	iTotalIdxWrite	:= iTotalIdxWrite + 1;

	IF tyParameter.tyAvl.bQueryId = TRUE THEN
		pa_tyXMLTable[iTotalIdxWrite].sTitle	:= 'AT';
		pa_tyXMLTable[iTotalIdxWrite].sValue	:= 'QueryId';
		pa_tyXMLTable[iTotalIdxWrite].uiSize	:= LEN(pa_tyXMLTable[iTotalIdxWrite].sValue);

		iTotalIdxWrite	:= iTotalIdxWrite + 1;

		pa_tyXMLTable[iTotalIdxWrite].sTitle	:= 'AV';
		pa_tyXMLTable[iTotalIdxWrite].sValue	:= tyParameter.tyData.sQueryId;
		pa_tyXMLTable[iTotalIdxWrite].uiSize	:= LEN(pa_tyXMLTable[iTotalIdxWrite].sValue);

		iTotalIdxWrite	:= iTotalIdxWrite + 1;
	END_IF

	IF tyParameter.tyAvl.bMachineId = TRUE THEN
		pa_tyXMLTable[iTotalIdxWrite].sTitle	:= 'AT';
		pa_tyXMLTable[iTotalIdxWrite].sValue	:= 'MachineId';
		pa_tyXMLTable[iTotalIdxWrite].uiSize	:= LEN(pa_tyXMLTable[iTotalIdxWrite].sValue);

		iTotalIdxWrite	:= iTotalIdxWrite + 1;

		pa_tyXMLTable[iTotalIdxWrite].sTitle	:= 'AV';
		pa_tyXMLTable[iTotalIdxWrite].sValue	:= tyParameter.tyData.sMachineId;
		pa_tyXMLTable[iTotalIdxWrite].uiSize	:= LEN(pa_tyXMLTable[iTotalIdxWrite].sValue);

		iTotalIdxWrite	:= iTotalIdxWrite + 1;
	END_IF

	IF tyParameter.tyAvl.bMagazineId = TRUE THEN
		pa_tyXMLTable[iTotalIdxWrite].sTitle	:= 'AT';
		pa_tyXMLTable[iTotalIdxWrite].sValue	:= 'MagazineId';
		pa_tyXMLTable[iTotalIdxWrite].uiSize	:= LEN(pa_tyXMLTable[iTotalIdxWrite].sValue);

		iTotalIdxWrite	:= iTotalIdxWrite + 1;

		pa_tyXMLTable[iTotalIdxWrite].sTitle	:= 'AV';
		pa_tyXMLTable[iTotalIdxWrite].sValue	:= tyParameter.tyData.sMagazineId;
		pa_tyXMLTable[iTotalIdxWrite].uiSize	:= LEN(pa_tyXMLTable[iTotalIdxWrite].sValue);

		iTotalIdxWrite	:= iTotalIdxWrite + 1;
	END_IF

	IF tyParameter.tyAvl.bSlotId = TRUE THEN
		pa_tyXMLTable[iTotalIdxWrite].sTitle	:= 'AT';
		pa_tyXMLTable[iTotalIdxWrite].sValue	:= 'SlotId';
		pa_tyXMLTable[iTotalIdxWrite].uiSize	:= LEN(pa_tyXMLTable[iTotalIdxWrite].sValue);

		iTotalIdxWrite	:= iTotalIdxWrite + 1;

		pa_tyXMLTable[iTotalIdxWrite].sTitle	:= 'AV';
		pa_tyXMLTable[iTotalIdxWrite].sValue	:= INT_TO_STRING(tyParameter.tyData.iSlotId);
		pa_tyXMLTable[iTotalIdxWrite].uiSize	:= LEN(pa_tyXMLTable[iTotalIdxWrite].sValue);

		iTotalIdxWrite	:= iTotalIdxWrite + 1;
	END_IF

	IF tyParameter.tyAvl.bBarcode = TRUE THEN
		pa_tyXMLTable[iTotalIdxWrite].sTitle	:= 'AT';
		pa_tyXMLTable[iTotalIdxWrite].sValue	:= 'Barcode';
		pa_tyXMLTable[iTotalIdxWrite].uiSize	:= LEN(pa_tyXMLTable[iTotalIdxWrite].sValue);

		iTotalIdxWrite	:= iTotalIdxWrite + 1;

		pa_tyXMLTable[iTotalIdxWrite].sTitle	:= 'AV';
		pa_tyXMLTable[iTotalIdxWrite].sValue	:= tyParameter.tyData.sBarcode;
		pa_tyXMLTable[iTotalIdxWrite].uiSize	:= LEN(pa_tyXMLTable[iTotalIdxWrite].sValue);

		iTotalIdxWrite	:= iTotalIdxWrite + 1;
	END_IF

	pa_tyXMLTable[iTotalIdxWrite].sTitle	:= 'ES';
	pa_tyXMLTable[iTotalIdxWrite].sValue	:= '';
	pa_tyXMLTable[iTotalIdxWrite].uiSize	:= LEN(pa_tyXMLTable[iTotalIdxWrite].sValue);

	iTotalIdxWrite	:= iTotalIdxWrite + 1;

	pa_tyXMLTable[iTotalIdxWrite].sTitle	:= 'ET';
	pa_tyXMLTable[iTotalIdxWrite].sValue	:= 'Hermes';
	pa_tyXMLTable[iTotalIdxWrite].uiSize	:= LEN(pa_tyXMLTable[iTotalIdxWrite].sValue);

	iTotalIdxWrite	:= iTotalIdxWrite + 1;

	pa_tyXMLTable[iTotalIdxWrite].sTitle	:= 'EN';
	pa_tyXMLTable[iTotalIdxWrite].sValue	:= '';
	pa_tyXMLTable[iTotalIdxWrite].uiSize	:= LEN(pa_tyXMLTable[iTotalIdxWrite].sValue);

	iTotalIdxWrite	:= iTotalIdxWrite + 1;

	iTotalIdxWrite	:= fHermesFormQueryWorkOrderInfo;

END_FUNCTION
```

#### fHermesFormSendWorkOrderInfo.st
```iecst
(* Hermes Form Send Work Order Info Table Data (Total Index Written In Table) *)
FUNCTION fHermesFormSendWorkOrderInfo

	memset(ADR(pa_tyXMLTable) , 0 , SIZEOF(pa_tyXMLTable));
	iTotalIdxWrite	:= 0;

	fHermesGetTimestamp(ADR(sTimestamp) , tyDTStructure);

	pa_tyXMLTable[iTotalIdxWrite].sTitle	:= 'ST';
	pa_tyXMLTable[iTotalIdxWrite].sValue	:= 'Hermes';
	pa_tyXMLTable[iTotalIdxWrite].uiSize	:= LEN(pa_tyXMLTable[iTotalIdxWrite].sValue);

	iTotalIdxWrite	:= iTotalIdxWrite + 1;

	pa_tyXMLTable[iTotalIdxWrite].sTitle	:= 'AT';
	pa_tyXMLTable[iTotalIdxWrite].sValue	:= 'Timestamp';
	pa_tyXMLTable[iTotalIdxWrite].uiSize	:= LEN(pa_tyXMLTable[iTotalIdxWrite].sValue);

	iTotalIdxWrite	:= iTotalIdxWrite + 1;

	pa_tyXMLTable[iTotalIdxWrite].sTitle	:= 'AV';
	pa_tyXMLTable[iTotalIdxWrite].sValue	:= sTimestamp;
	pa_tyXMLTable[iTotalIdxWrite].uiSize	:= LEN(pa_tyXMLTable[iTotalIdxWrite].sValue);

	iTotalIdxWrite	:= iTotalIdxWrite + 1;

	pa_tyXMLTable[iTotalIdxWrite].sTitle	:= 'EN';
	pa_tyXMLTable[iTotalIdxWrite].sValue	:= '';
	pa_tyXMLTable[iTotalIdxWrite].uiSize	:= LEN(pa_tyXMLTable[iTotalIdxWrite].sValue);

	iTotalIdxWrite	:= iTotalIdxWrite + 1;

	pa_tyXMLTable[iTotalIdxWrite].sTitle	:= 'ST';
	pa_tyXMLTable[iTotalIdxWrite].sValue	:= 'SendWorkOrderInfo';
	pa_tyXMLTable[iTotalIdxWrite].uiSize	:= LEN(pa_tyXMLTable[iTotalIdxWrite].sValue);

	iTotalIdxWrite	:= iTotalIdxWrite + 1;

	IF tyParameter.tyAvl.bQueryId = TRUE THEN
		pa_tyXMLTable[iTotalIdxWrite].sTitle	:= 'AT';
		pa_tyXMLTable[iTotalIdxWrite].sValue	:= 'QueryId';
		pa_tyXMLTable[iTotalIdxWrite].uiSize	:= LEN(pa_tyXMLTable[iTotalIdxWrite].sValue);

		iTotalIdxWrite	:= iTotalIdxWrite + 1;

		pa_tyXMLTable[iTotalIdxWrite].sTitle	:= 'AV';
		pa_tyXMLTable[iTotalIdxWrite].sValue	:= tyParameter.tyData.sQueryId;
		pa_tyXMLTable[iTotalIdxWrite].uiSize	:= LEN(pa_tyXMLTable[iTotalIdxWrite].sValue);

		iTotalIdxWrite	:= iTotalIdxWrite + 1;
	END_IF

	IF tyParameter.tyAvl.bWorkOrderId = TRUE THEN
		pa_tyXMLTable[iTotalIdxWrite].sTitle	:= 'AT';
		pa_tyXMLTable[iTotalIdxWrite].sValue	:= 'WorkOrderId';
		pa_tyXMLTable[iTotalIdxWrite].uiSize	:= LEN(pa_tyXMLTable[iTotalIdxWrite].sValue);

		iTotalIdxWrite	:= iTotalIdxWrite + 1;

		pa_tyXMLTable[iTotalIdxWrite].sTitle	:= 'AV';
		pa_tyXMLTable[iTotalIdxWrite].sValue	:= tyParameter.tyData.sWorkOrderId;
		pa_tyXMLTable[iTotalIdxWrite].uiSize	:= LEN(pa_tyXMLTable[iTotalIdxWrite].sValue);

		iTotalIdxWrite	:= iTotalIdxWrite + 1;
	END_IF

	IF tyParameter.tyAvl.bBatchId = TRUE THEN
		pa_tyXMLTable[iTotalIdxWrite].sTitle	:= 'AT';
		pa_tyXMLTable[iTotalIdxWrite].sValue	:= 'BatchId';
		pa_tyXMLTable[iTotalIdxWrite].uiSize	:= LEN(pa_tyXMLTable[iTotalIdxWrite].sValue);

		iTotalIdxWrite	:= iTotalIdxWrite + 1;

		pa_tyXMLTable[iTotalIdxWrite].sTitle	:= 'AV';
		pa_tyXMLTable[iTotalIdxWrite].sValue	:= tyParameter.tyData.sBatchId;
		pa_tyXMLTable[iTotalIdxWrite].uiSize	:= LEN(pa_tyXMLTable[iTotalIdxWrite].sValue);

		iTotalIdxWrite	:= iTotalIdxWrite + 1;
	END_IF

	IF tyParameter.tyAvl.bBoardId = TRUE THEN
		pa_tyXMLTable[iTotalIdxWrite].sTitle	:= 'AT';
		pa_tyXMLTable[iTotalIdxWrite].sValue	:= 'BoardId';
		pa_tyXMLTable[iTotalIdxWrite].uiSize	:= LEN(pa_tyXMLTable[iTotalIdxWrite].sValue);

		iTotalIdxWrite	:= iTotalIdxWrite + 1;

		pa_tyXMLTable[iTotalIdxWrite].sTitle	:= 'AV';
		pa_tyXMLTable[iTotalIdxWrite].sValue	:= tyParameter.tyData.sBoardId;
		pa_tyXMLTable[iTotalIdxWrite].uiSize	:= LEN(pa_tyXMLTable[iTotalIdxWrite].sValue);

		iTotalIdxWrite	:= iTotalIdxWrite + 1;
	END_IF

	IF tyParameter.tyAvl.bBoardIdCreatedBy = TRUE THEN
		pa_tyXMLTable[iTotalIdxWrite].sTitle	:= 'AT';
		pa_tyXMLTable[iTotalIdxWrite].sValue	:= 'BoardIdCreatedBy';
		pa_tyXMLTable[iTotalIdxWrite].uiSize	:= LEN(pa_tyXMLTable[iTotalIdxWrite].sValue);

		iTotalIdxWrite	:= iTotalIdxWrite + 1;

		pa_tyXMLTable[iTotalIdxWrite].sTitle	:= 'AV';
		pa_tyXMLTable[iTotalIdxWrite].sValue	:= tyParameter.tyData.sBoardIdCreatedBy;
		pa_tyXMLTable[iTotalIdxWrite].uiSize	:= LEN(pa_tyXMLTable[iTotalIdxWrite].sValue);

		iTotalIdxWrite	:= iTotalIdxWrite + 1;
	END_IF

	IF tyParameter.tyAvl.bFailedBoard = TRUE THEN
		pa_tyXMLTable[iTotalIdxWrite].sTitle	:= 'AT';
		pa_tyXMLTable[iTotalIdxWrite].sValue	:= 'FailedBoard';
		pa_tyXMLTable[iTotalIdxWrite].uiSize	:= LEN(pa_tyXMLTable[iTotalIdxWrite].sValue);

		iTotalIdxWrite	:= iTotalIdxWrite + 1;

		pa_tyXMLTable[iTotalIdxWrite].sTitle	:= 'AV';
		pa_tyXMLTable[iTotalIdxWrite].sValue	:= DINT_TO_STRING(UDINT_TO_DINT(tyParameter.tyData.eFailedBoard));
		pa_tyXMLTable[iTotalIdxWrite].uiSize	:= LEN(pa_tyXMLTable[iTotalIdxWrite].sValue);

		iTotalIdxWrite	:= iTotalIdxWrite + 1;
	END_IF

	IF tyParameter.tyAvl.bProductTypeId = TRUE THEN
		pa_tyXMLTable[iTotalIdxWrite].sTitle	:= 'AT';
		pa_tyXMLTable[iTotalIdxWrite].sValue	:= 'ProductTypeId';
		pa_tyXMLTable[iTotalIdxWrite].uiSize	:= LEN(pa_tyXMLTable[iTotalIdxWrite].sValue);

		iTotalIdxWrite	:= iTotalIdxWrite + 1;

		pa_tyXMLTable[iTotalIdxWrite].sTitle	:= 'AV';
		pa_tyXMLTable[iTotalIdxWrite].sValue	:= tyParameter.tyData.sProductTypeId;
		pa_tyXMLTable[iTotalIdxWrite].uiSize	:= LEN(pa_tyXMLTable[iTotalIdxWrite].sValue);

		iTotalIdxWrite	:= iTotalIdxWrite + 1;
	END_IF

	IF tyParameter.tyAvl.bFlippedBoard = TRUE THEN
		pa_tyXMLTable[iTotalIdxWrite].sTitle	:= 'AT';
		pa_tyXMLTable[iTotalIdxWrite].sValue	:= 'FlippedBoard';
		pa_tyXMLTable[iTotalIdxWrite].uiSize	:= LEN(pa_tyXMLTable[iTotalIdxWrite].sValue);

		iTotalIdxWrite	:= iTotalIdxWrite + 1;

		pa_tyXMLTable[iTotalIdxWrite].sTitle	:= 'AV';
		pa_tyXMLTable[iTotalIdxWrite].sValue	:= DINT_TO_STRING(UDINT_TO_DINT(tyParameter.tyData.eFlippedBoard));
		pa_tyXMLTable[iTotalIdxWrite].uiSize	:= LEN(pa_tyXMLTable[iTotalIdxWrite].sValue);

		iTotalIdxWrite	:= iTotalIdxWrite + 1;
	END_IF

	IF tyParameter.tyAvl.bTopBarcode = TRUE THEN
		pa_tyXMLTable[iTotalIdxWrite].sTitle	:= 'AT';
		pa_tyXMLTable[iTotalIdxWrite].sValue	:= 'TopBarcode';
		pa_tyXMLTable[iTotalIdxWrite].uiSize	:= LEN(pa_tyXMLTable[iTotalIdxWrite].sValue);

		iTotalIdxWrite	:= iTotalIdxWrite + 1;

		pa_tyXMLTable[iTotalIdxWrite].sTitle	:= 'AV';
		pa_tyXMLTable[iTotalIdxWrite].sValue	:= tyParameter.tyData.sTopBarcode;
		pa_tyXMLTable[iTotalIdxWrite].uiSize	:= LEN(pa_tyXMLTable[iTotalIdxWrite].sValue);

		iTotalIdxWrite	:= iTotalIdxWrite + 1;
	END_IF

	IF tyParameter.tyAvl.bBottomBarcode = TRUE THEN
		pa_tyXMLTable[iTotalIdxWrite].sTitle	:= 'AT';
		pa_tyXMLTable[iTotalIdxWrite].sValue	:= 'BottomBarcode';
		pa_tyXMLTable[iTotalIdxWrite].uiSize	:= LEN(pa_tyXMLTable[iTotalIdxWrite].sValue);

		iTotalIdxWrite	:= iTotalIdxWrite + 1;

		pa_tyXMLTable[iTotalIdxWrite].sTitle	:= 'AV';
		pa_tyXMLTable[iTotalIdxWrite].sValue	:= tyParameter.tyData.sBottomBarcode;
		pa_tyXMLTable[iTotalIdxWrite].uiSize	:= LEN(pa_tyXMLTable[iTotalIdxWrite].sValue);

		iTotalIdxWrite	:= iTotalIdxWrite + 1;
	END_IF

	IF tyParameter.tyAvl.bLength = TRUE THEN
		pa_tyXMLTable[iTotalIdxWrite].sTitle	:= 'AT';
		pa_tyXMLTable[iTotalIdxWrite].sValue	:= 'Length';
		pa_tyXMLTable[iTotalIdxWrite].uiSize	:= LEN(pa_tyXMLTable[iTotalIdxWrite].sValue);

		iTotalIdxWrite	:= iTotalIdxWrite + 1;

		pa_tyXMLTable[iTotalIdxWrite].sTitle	:= 'AV';
		pa_tyXMLTable[iTotalIdxWrite].sValue	:= REAL_TO_STRING(tyParameter.tyData.rLength);
		pa_tyXMLTable[iTotalIdxWrite].uiSize	:= LEN(pa_tyXMLTable[iTotalIdxWrite].sValue);

		iTotalIdxWrite	:= iTotalIdxWrite + 1;
	END_IF

	IF tyParameter.tyAvl.bWidth = TRUE THEN
		pa_tyXMLTable[iTotalIdxWrite].sTitle	:= 'AT';
		pa_tyXMLTable[iTotalIdxWrite].sValue	:= 'Width';
		pa_tyXMLTable[iTotalIdxWrite].uiSize	:= LEN(pa_tyXMLTable[iTotalIdxWrite].sValue);

		iTotalIdxWrite	:= iTotalIdxWrite + 1;

		pa_tyXMLTable[iTotalIdxWrite].sTitle	:= 'AV';
		pa_tyXMLTable[iTotalIdxWrite].sValue	:= REAL_TO_STRING(tyParameter.tyData.rWidth);
		pa_tyXMLTable[iTotalIdxWrite].uiSize	:= LEN(pa_tyXMLTable[iTotalIdxWrite].sValue);

		iTotalIdxWrite	:= iTotalIdxWrite + 1;
	END_IF

	IF tyParameter.tyAvl.bThickness = TRUE THEN
		pa_tyXMLTable[iTotalIdxWrite].sTitle	:= 'AT';
		pa_tyXMLTable[iTotalIdxWrite].sValue	:= 'Thickness';
		pa_tyXMLTable[iTotalIdxWrite].uiSize	:= LEN(pa_tyXMLTable[iTotalIdxWrite].sValue);

		iTotalIdxWrite	:= iTotalIdxWrite + 1;

		pa_tyXMLTable[iTotalIdxWrite].sTitle	:= 'AV';
		pa_tyXMLTable[iTotalIdxWrite].sValue	:= REAL_TO_STRING(tyParameter.tyData.rThickness);
		pa_tyXMLTable[iTotalIdxWrite].uiSize	:= LEN(pa_tyXMLTable[iTotalIdxWrite].sValue);

		iTotalIdxWrite	:= iTotalIdxWrite + 1;
	END_IF

	IF tyParameter.tyAvl.bConveyorSpeed = TRUE THEN
		pa_tyXMLTable[iTotalIdxWrite].sTitle	:= 'AT';
		pa_tyXMLTable[iTotalIdxWrite].sValue	:= 'ConveyorSpeed';
		pa_tyXMLTable[iTotalIdxWrite].uiSize	:= LEN(pa_tyXMLTable[iTotalIdxWrite].sValue);

		iTotalIdxWrite	:= iTotalIdxWrite + 1;

		pa_tyXMLTable[iTotalIdxWrite].sTitle	:= 'AV';
		pa_tyXMLTable[iTotalIdxWrite].sValue	:= REAL_TO_STRING(tyParameter.tyData.rConveyorSpeed);
		pa_tyXMLTable[iTotalIdxWrite].uiSize	:= LEN(pa_tyXMLTable[iTotalIdxWrite].sValue);

		iTotalIdxWrite	:= iTotalIdxWrite + 1;
	END_IF

	IF tyParameter.tyAvl.bTopClearanceHeight = TRUE THEN
		pa_tyXMLTable[iTotalIdxWrite].sTitle	:= 'AT';
		pa_tyXMLTable[iTotalIdxWrite].sValue	:= 'TopClearanceHeight';
		pa_tyXMLTable[iTotalIdxWrite].uiSize	:= LEN(pa_tyXMLTable[iTotalIdxWrite].sValue);

		iTotalIdxWrite	:= iTotalIdxWrite + 1;

		pa_tyXMLTable[iTotalIdxWrite].sTitle	:= 'AV';
		pa_tyXMLTable[iTotalIdxWrite].sValue	:= REAL_TO_STRING(tyParameter.tyData.rTopClearanceHeight);
		pa_tyXMLTable[iTotalIdxWrite].uiSize	:= LEN(pa_tyXMLTable[iTotalIdxWrite].sValue);

		iTotalIdxWrite	:= iTotalIdxWrite + 1;
	END_IF

	IF tyParameter.tyAvl.bBottomClearanceHeight = TRUE THEN
		pa_tyXMLTable[iTotalIdxWrite].sTitle	:= 'AT';
		pa_tyXMLTable[iTotalIdxWrite].sValue	:= 'BottomClearanceHeight';
		pa_tyXMLTable[iTotalIdxWrite].uiSize	:= LEN(pa_tyXMLTable[iTotalIdxWrite].sValue);

		iTotalIdxWrite	:= iTotalIdxWrite + 1;

		pa_tyXMLTable[iTotalIdxWrite].sTitle	:= 'AV';
		pa_tyXMLTable[iTotalIdxWrite].sValue	:= REAL_TO_STRING(tyParameter.tyData.rBottomClearanceHeight);
		pa_tyXMLTable[iTotalIdxWrite].uiSize	:= LEN(pa_tyXMLTable[iTotalIdxWrite].sValue);

		iTotalIdxWrite	:= iTotalIdxWrite + 1;
	END_IF

	IF tyParameter.tyAvl.bWeight = TRUE THEN
		pa_tyXMLTable[iTotalIdxWrite].sTitle	:= 'AT';
		pa_tyXMLTable[iTotalIdxWrite].sValue	:= 'Weight';
		pa_tyXMLTable[iTotalIdxWrite].uiSize	:= LEN(pa_tyXMLTable[iTotalIdxWrite].sValue);

		iTotalIdxWrite	:= iTotalIdxWrite + 1;

		pa_tyXMLTable[iTotalIdxWrite].sTitle	:= 'AV';
		pa_tyXMLTable[iTotalIdxWrite].sValue	:= REAL_TO_STRING(tyParameter.tyData.rWeight);
		pa_tyXMLTable[iTotalIdxWrite].uiSize	:= LEN(pa_tyXMLTable[iTotalIdxWrite].sValue);

		iTotalIdxWrite	:= iTotalIdxWrite + 1;
	END_IF

	IF tyParameter.tyAvl.bRoute = TRUE THEN
		pa_tyXMLTable[iTotalIdxWrite].sTitle	:= 'AT';
		pa_tyXMLTable[iTotalIdxWrite].sValue	:= 'Route';
		pa_tyXMLTable[iTotalIdxWrite].uiSize	:= LEN(pa_tyXMLTable[iTotalIdxWrite].sValue);

		iTotalIdxWrite	:= iTotalIdxWrite + 1;

		pa_tyXMLTable[iTotalIdxWrite].sTitle	:= 'AV';
		pa_tyXMLTable[iTotalIdxWrite].sValue	:= INT_TO_STRING(tyParameter.tyData.iRoute);
		pa_tyXMLTable[iTotalIdxWrite].uiSize	:= LEN(pa_tyXMLTable[iTotalIdxWrite].sValue);

		iTotalIdxWrite	:= iTotalIdxWrite + 1;
	END_IF

	pa_tyXMLTable[iTotalIdxWrite].sTitle	:= 'ES';
	pa_tyXMLTable[iTotalIdxWrite].sValue	:= '';
	pa_tyXMLTable[iTotalIdxWrite].uiSize	:= LEN(pa_tyXMLTable[iTotalIdxWrite].sValue);

	iTotalIdxWrite	:= iTotalIdxWrite + 1;

	pa_tyXMLTable[iTotalIdxWrite].sTitle	:= 'ET';
	pa_tyXMLTable[iTotalIdxWrite].sValue	:= 'Hermes';
	pa_tyXMLTable[iTotalIdxWrite].uiSize	:= LEN(pa_tyXMLTable[iTotalIdxWrite].sValue);

	iTotalIdxWrite	:= iTotalIdxWrite + 1;

	pa_tyXMLTable[iTotalIdxWrite].sTitle	:= 'EN';
	pa_tyXMLTable[iTotalIdxWrite].sValue	:= '';
	pa_tyXMLTable[iTotalIdxWrite].uiSize	:= LEN(pa_tyXMLTable[iTotalIdxWrite].sValue);

	iTotalIdxWrite	:= iTotalIdxWrite + 1;

	iTotalIdxWrite	:= fHermesFormSendWorkOrderInfo;

END_FUNCTION
```

#### fHermesFormCommand.st
```iecst
(* Hermes Form Query Board Info Table Data (Total Index Written In Table) *)
FUNCTION fHermesFormCommand

	memset(ADR(pa_tyXMLTable) , 0 , SIZEOF(pa_tyXMLTable));
	iTotalIdxWrite	:= 0;

	fHermesGetTimestamp(ADR(sTimestamp) , tyDTStructure);

	pa_tyXMLTable[iTotalIdxWrite].sTitle	:= 'ST';
	pa_tyXMLTable[iTotalIdxWrite].sValue	:= 'Hermes';
	pa_tyXMLTable[iTotalIdxWrite].uiSize	:= LEN(pa_tyXMLTable[iTotalIdxWrite].sValue);

	iTotalIdxWrite	:= iTotalIdxWrite + 1;

	pa_tyXMLTable[iTotalIdxWrite].sTitle	:= 'AT';
	pa_tyXMLTable[iTotalIdxWrite].sValue	:= 'Timestamp';
	pa_tyXMLTable[iTotalIdxWrite].uiSize	:= LEN(pa_tyXMLTable[iTotalIdxWrite].sValue);

	iTotalIdxWrite	:= iTotalIdxWrite + 1;

	pa_tyXMLTable[iTotalIdxWrite].sTitle	:= 'AV';
	pa_tyXMLTable[iTotalIdxWrite].sValue	:= sTimestamp;
	pa_tyXMLTable[iTotalIdxWrite].uiSize	:= LEN(pa_tyXMLTable[iTotalIdxWrite].sValue);

	iTotalIdxWrite	:= iTotalIdxWrite + 1;

	pa_tyXMLTable[iTotalIdxWrite].sTitle	:= 'EN';
	pa_tyXMLTable[iTotalIdxWrite].sValue	:= '';
	pa_tyXMLTable[iTotalIdxWrite].uiSize	:= LEN(pa_tyXMLTable[iTotalIdxWrite].sValue);

	iTotalIdxWrite	:= iTotalIdxWrite + 1;

	pa_tyXMLTable[iTotalIdxWrite].sTitle	:= 'ST';
	pa_tyXMLTable[iTotalIdxWrite].sValue	:= 'Command';
	pa_tyXMLTable[iTotalIdxWrite].uiSize	:= LEN(pa_tyXMLTable[iTotalIdxWrite].sValue);

	iTotalIdxWrite	:= iTotalIdxWrite + 1;

	IF tyParameter.tyAvl.bCommand = TRUE THEN
		pa_tyXMLTable[iTotalIdxWrite].sTitle	:= 'AT';
		pa_tyXMLTable[iTotalIdxWrite].sValue	:= 'Command';
		pa_tyXMLTable[iTotalIdxWrite].uiSize	:= LEN(pa_tyXMLTable[iTotalIdxWrite].sValue);

		iTotalIdxWrite	:= iTotalIdxWrite + 1;

		pa_tyXMLTable[iTotalIdxWrite].sTitle	:= 'AV';
		pa_tyXMLTable[iTotalIdxWrite].sValue	:= INT_TO_STRING(UDINT_TO_INT(tyParameter.tyData.eCommand));
		pa_tyXMLTable[iTotalIdxWrite].uiSize	:= LEN(pa_tyXMLTable[iTotalIdxWrite].sValue);

		iTotalIdxWrite	:= iTotalIdxWrite + 1;
	END_IF

	pa_tyXMLTable[iTotalIdxWrite].sTitle	:= 'ES';
	pa_tyXMLTable[iTotalIdxWrite].sValue	:= '';
	pa_tyXMLTable[iTotalIdxWrite].uiSize	:= LEN(pa_tyXMLTable[iTotalIdxWrite].sValue);

	iTotalIdxWrite	:= iTotalIdxWrite + 1;

	pa_tyXMLTable[iTotalIdxWrite].sTitle	:= 'ET';
	pa_tyXMLTable[iTotalIdxWrite].sValue	:= 'Hermes';
	pa_tyXMLTable[iTotalIdxWrite].uiSize	:= LEN(pa_tyXMLTable[iTotalIdxWrite].sValue);

	iTotalIdxWrite	:= iTotalIdxWrite + 1;

	pa_tyXMLTable[iTotalIdxWrite].sTitle	:= 'EN';
	pa_tyXMLTable[iTotalIdxWrite].sValue	:= '';
	pa_tyXMLTable[iTotalIdxWrite].uiSize	:= LEN(pa_tyXMLTable[iTotalIdxWrite].sValue);

	iTotalIdxWrite	:= iTotalIdxWrite + 1;

	iTotalIdxWrite	:= fHermesFormCommand;

END_FUNCTION
```

#### fHermesChkParamBAMR.st
```iecst
(* Hermes Checking Parameter Board Available & Machine Ready *)
FUNCTION fHermesChkParamBAMR

	fHermesChkParamBAMR	:= 0;

	IF fHermesChkParamBAMR = 0 THEN

		IF tyBoardAvailable.tyAvl.bBoardId = TRUE AND tyMachineReady.tyAvl.bBoardId = TRUE THEN

			IF tyBoardAvailable.tyData.sBoardId <> tyMachineReady.tyData.sBoardId THEN

				fHermesChkParamBAMR	:= 2700;	//BoardId Mismatch While Checking Board Available & Machine Ready

			END_IF

		END_IF

	END_IF

	IF fHermesChkParamBAMR = 0 THEN

		IF tyBoardAvailable.tyAvl.bProductTypeId = TRUE AND tyMachineReady.tyAvl.bProductTypeId = TRUE THEN

			IF tyBoardAvailable.tyData.sProductTypeId <> tyMachineReady.tyData.sProductTypeId THEN

				fHermesChkParamBAMR	:= 2701;	//ProductTypeId Mismatch While Checking Board Available & Machine Ready

			END_IF

		END_IF

	END_IF

	IF fHermesChkParamBAMR = 0 THEN

		IF tyBoardAvailable.tyAvl.bFlippedBoard = TRUE AND tyMachineReady.tyAvl.bFlippedBoard = TRUE THEN

			IF tyBoardAvailable.tyData.eFlippedBoard <> tyMachineReady.tyData.eFlippedBoard THEN

				fHermesChkParamBAMR	:= 2702;	//FlippedBoard Mismatch While Checking Board Available & Machine Ready

			END_IF

		END_IF

	END_IF

	IF fHermesChkParamBAMR = 0 THEN

		IF tyBoardAvailable.tyAvl.bLength = TRUE AND tyMachineReady.tyAvl.bLength = TRUE THEN

			IF tyBoardAvailable.tyData.rLength <> tyMachineReady.tyData.rLength THEN

				fHermesChkParamBAMR	:= 2703;	//Length Mismatch While Checking Board Available & Machine Ready

			END_IF

		END_IF

	END_IF

	IF fHermesChkParamBAMR = 0 THEN

		IF tyBoardAvailable.tyAvl.bWidth = TRUE AND tyMachineReady.tyAvl.bWidth = TRUE THEN

			IF tyBoardAvailable.tyData.rWidth <> tyMachineReady.tyData.rWidth THEN

				fHermesChkParamBAMR	:= 2704;	//Width Mismatch While Checking Board Available & Machine Ready

			END_IF

		END_IF

	END_IF

	IF fHermesChkParamBAMR = 0 THEN

		IF tyBoardAvailable.tyAvl.bThickness = TRUE AND tyMachineReady.tyAvl.bThickness = TRUE THEN

			IF tyBoardAvailable.tyData.rThickness <> tyMachineReady.tyData.rThickness THEN

				fHermesChkParamBAMR	:= 2705;	//Thickness Mismatch While Checking Board Available & Machine Ready

			END_IF

		END_IF

	END_IF

	IF fHermesChkParamBAMR = 0 THEN

		IF tyBoardAvailable.tyAvl.bConveyorSpeed = TRUE AND tyMachineReady.tyAvl.bConveyorSpeed = TRUE THEN

			IF tyBoardAvailable.tyData.rConveyorSpeed <> tyMachineReady.tyData.rConveyorSpeed THEN

				fHermesChkParamBAMR	:= 2706;	//ConveyorSpeed Mismatch While Checking Board Available & Machine Ready

			END_IF

		END_IF

	END_IF

	IF fHermesChkParamBAMR = 0 THEN

		IF tyBoardAvailable.tyAvl.bTopClearanceHeight = TRUE AND tyMachineReady.tyAvl.bTopClearanceHeight = TRUE THEN

			IF tyBoardAvailable.tyData.rTopClearanceHeight <> tyMachineReady.tyData.rTopClearanceHeight THEN

				fHermesChkParamBAMR	:= 2707;	//TopClearanceHeight Mismatch While Checking Board Available & Machine Ready

			END_IF

		END_IF

	END_IF

	IF fHermesChkParamBAMR = 0 THEN

		IF tyBoardAvailable.tyAvl.bBottomClearanceHeight = TRUE AND tyMachineReady.tyAvl.bBottomClearanceHeight = TRUE THEN

			IF tyBoardAvailable.tyData.rBottomClearanceHeight <> tyMachineReady.tyData.rBottomClearanceHeight THEN

				fHermesChkParamBAMR	:= 2708;	//BottomClearanceHeight Mismatch While Checking Board Available & Machine Ready

			END_IF

		END_IF

	END_IF

	IF fHermesChkParamBAMR = 0 THEN

		IF tyBoardAvailable.tyAvl.bWeight = TRUE AND tyMachineReady.tyAvl.bWeight = TRUE THEN

			IF tyBoardAvailable.tyData.rWeight <> tyMachineReady.tyData.rWeight THEN

				fHermesChkParamBAMR	:= 2709;	//Weight Mismatch While Checking Board Available & Machine Ready

			END_IF

		END_IF

	END_IF

END_FUNCTION
```

#### fHermesChkParamBAST.st
```iecst
(* Hermes Checking Parameter Board Available & Start Transport *)
FUNCTION fHermesChkParamBAST

	fHermesChkParamBAST	:= 0;

	IF tyBoardAvailable.tyAvl.bBoardId = TRUE AND tyStartTransport.tyAvl.bBoardId = TRUE THEN

		IF tyBoardAvailable.tyData.sBoardId <> tyStartTransport.tyData.sBoardId THEN

			fHermesChkParamBAST	:= 2710;	//BoardId Mismatch While Checking Board Available & Start Transport

		END_IF

	ELSE

		fHermesChkParamBAST	:= 2711;	//BoardId Missing While Checking Board Available & Start Transport

	END_IF

END_FUNCTION
```

#### fHermesChkParamSTST.st
```iecst
(* Hermes Checking Parameter Start Transport & Stop Transport *)
FUNCTION fHermesChkParamSTST

	fHermesChkParamSTST	:= 0;

	IF tyStartTransport.tyAvl.bBoardId = TRUE AND tyStopTransport.tyAvl.bBoardId = TRUE THEN

		IF tyStartTransport.tyData.sBoardId <> tyStopTransport.tyData.sBoardId THEN

			fHermesChkParamSTST	:= 2712;	//BoardId Mismatch While Checking Start Transport & Stop Transport

		END_IF

	ELSE

		fHermesChkParamSTST	:= 2713;	//BoardId Missing While Checking Start Transport & Stop Transport

	END_IF

END_FUNCTION
```

#### fHermesChkParamSTTF.st
```iecst
(* Hermes Checking Parameter Start Transport & Transport Finished *)
FUNCTION fHermesChkParamSTTF

	fHermesChkParamSTTF	:= 0;

	IF tyStartTransport.tyAvl.bBoardId = TRUE AND tyTransportFinished.tyAvl.bBoardId = TRUE THEN

		IF tyStartTransport.tyData.sBoardId <> tyTransportFinished.tyData.sBoardId THEN

			fHermesChkParamSTTF	:= 2714;	//BoardId Mismatch While Checking Start Transport & Transport Finished

		END_IF

	ELSE

		fHermesChkParamSTTF	:= 2715;	//BoardId Missing While Checking Start Transport & Transport Finished

	END_IF

END_FUNCTION
```

#### fHermesChkParamBFMR.st
```iecst
(* Hermes Checking Parameter Board Forecast & Machine Ready *)
FUNCTION fHermesChkParamBFMR

      fHermesChkParamBFMR :=0;

	    IF tyBoardForecast.tyData.sForecastId <> tyMachineReady.tyData.sForecastId THEN

				fHermesChkParamBFMR	:= 2716;	//ForecastId Mismatch While Checking Board Forecast & Machine Ready

		END_IF

		IF tyBoardForecast.tyAvl.bProductTypeId = TRUE AND tyMachineReady.tyAvl.bProductTypeId = TRUE THEN

			IF tyBoardForecast.tyData.sProductTypeId <> tyMachineReady.tyData.sProductTypeId THEN

					fHermesChkParamBFMR	:= 2717;	//ProductTypeId Mismatch While Checking Board Forecast & Machine Ready

			END_IF

		END_IF

		IF tyBoardForecast.tyAvl.bWidth = TRUE AND tyMachineReady.tyAvl.bWidth = TRUE THEN

			IF tyBoardForecast.tyData.rWidth <> tyMachineReady.tyData.rWidth THEN

				fHermesChkParamBFMR	:= 2718;	//Width Mismatch While Checking Board Forecast & Machine Ready

			END_IF

		END_IF

END_FUNCTION
```

#### fHermesChkParamSD.st
```iecst
(* Hermes Checking Parameter Service Description *)
FUNCTION fHermesChkParamSD

	fHermesChkParamSD	:= 0;

	IF fHermesChkParamSD = 0 THEN

		IF tyServiceDescription.tyAvl.bMachineId = FALSE THEN

			fHermesChkParamSD	:= 2727;	//MachineId Missing While Checking Service Description

		END_IF

	END_IF

	IF fHermesChkParamSD = 0 THEN

		IF tyServiceDescription.tyAvl.bLaneId = TRUE THEN

			IF tyServiceDescription.tyData.iLaneId <= 0 THEN

				fHermesChkParamSD	:= 2728;	//LandId Out Of Range While Checking Service Description

			ELSIF tyServiceDescription.tyData.iLaneId <> iLaneId THEN

				fHermesChkParamSD	:= 2726;	//LaneId Mismatch While Checking Service Description

			END_IF

		ELSE

			fHermesChkParamSD	:= 2729;	//LandId Missing While Checking Service Description

		END_IF

	END_IF

	IF fHermesChkParamSD = 0 THEN

		IF tyServiceDescription.tyAvl.bVersion = FALSE THEN

			fHermesChkParamSD	:= 2730;	//Version Missing While Checking Service Description

		END_IF

	END_IF

	IF fHermesChkParamSD = 0 THEN

		IF tyServiceDescription.tyAvl.bSupportedFeatures = FALSE THEN

			fHermesChkParamSD	:= 2731;	//SupportedFeatures Missing While Checking Service Description

		END_IF

	END_IF

END_FUNCTION
```

#### fHermesChkParamSSD.st
```iecst
(* Hermes Checking Parameter Supervisory Service Description *)
FUNCTION fHermesChkParamSSD

	fHermesChkParamSSD	:= 0;

	IF fHermesChkParamSSD = 0 THEN

		IF tyServiceDescription.tyAvl.bSystemId = FALSE THEN

			fHermesChkParamSSD	:= 2719;	//SystemId Missing While Checking Service Description

		END_IF

	END_IF

	IF fHermesChkParamSSD = 0 THEN

		IF tyServiceDescription.tyAvl.bVersion = FALSE THEN

			fHermesChkParamSSD	:= 2730;	//Version Missing While Checking Service Description

		END_IF

	END_IF

	IF fHermesChkParamSSD = 0 THEN

		IF tyServiceDescription.tyAvl.bSupportedFeatures = FALSE THEN

			fHermesChkParamSSD	:= 2731;	//SupportedFeatures Missing While Checking Service Description

		END_IF

	END_IF

END_FUNCTION
```

#### fHermesChkParamN.st
```iecst
(* Hermes Checking Parameter Notification *)
FUNCTION fHermesChkParamN

	fHermesChkParamN	:= 0;

	IF fHermesChkParamN = 0 THEN

		IF tyNotification.tyAvl.bNotificationCode = TRUE THEN

			IF tyNotification.tyData.iNotificationCode <= 0 THEN

				fHermesChkParamN	:= 2732;	//NotificationCode Out Of Range While Checking Notification

			END_IF

		ELSE

			fHermesChkParamN	:= 2733;	//NotificationCode Missing While Checking Notification

		END_IF

	END_IF

	IF fHermesChkParamN = 0 THEN

		IF tyNotification.tyAvl.bSeverity = FALSE THEN

			fHermesChkParamN	:= 2734;	//Severity Missing While Checking Notification

		END_IF

	END_IF

	IF fHermesChkParamN = 0 THEN

		IF tyNotification.tyAvl.bDescription = FALSE THEN

			fHermesChkParamN	:= 2735;	//Description Missing While Checking Notification

		END_IF

	END_IF

END_FUNCTION
```

#### fHermesChkParamBA.st
```iecst
(* Hermes Checking Parameter Board Available *)
FUNCTION fHermesChkParamBA

	fHermesChkParamBA	:= 0;

	IF fHermesChkParamBA = 0 THEN

		IF tyBoardAvailable.tyAvl.bBoardId = FALSE THEN

			fHermesChkParamBA	:= 2736;	//BoardId Missing While Checking Board Available

		END_IF

	END_IF

	IF fHermesChkParamBA = 0 THEN

		IF tyBoardAvailable.tyAvl.bBoardIdCreatedBy = FALSE THEN

			fHermesChkParamBA	:= 2737;	//BoardIdCreatedBy Missing While Checking Board Available

		END_IF

	END_IF

	IF fHermesChkParamBA = 0 THEN

		IF tyBoardAvailable.tyAvl.bFailedBoard = FALSE THEN

			fHermesChkParamBA	:= 2738;	//FailedBoard Missing While Checking Board Available

		END_IF

	END_IF

	IF fHermesChkParamBA = 0 THEN

		IF tyBoardAvailable.tyAvl.bFlippedBoard = FALSE THEN

			fHermesChkParamBA	:= 2739;	//FlippedBoard Missing While Checking Board Available

		END_IF

	END_IF

END_FUNCTION
```

#### fHermesChkParamMR.st
```iecst
(* Hermes Checking Parameter Machine Ready *)
FUNCTION fHermesChkParamMR

	fHermesChkParamMR	:= 0;

	IF fHermesChkParamMR = 0 THEN

		IF tyMachineReady.tyAvl.bFailedBoard = FALSE THEN

			fHermesChkParamMR	:= 2740;	//FailedBoard Missing While Checking Machine Ready

		END_IF

	END_IF

END_FUNCTION
```

#### fHermesChkParamSAT.st
```iecst
(* Hermes Checking Parameter Start Transport *)
FUNCTION fHermesChkParamSAT

	fHermesChkParamSAT	:= 0;

	IF fHermesChkParamSAT = 0 THEN

		IF tyStartTransport.tyAvl.bBoardId = FALSE THEN

			fHermesChkParamSAT	:= 2741;	//BoardId Missing While Checking Start Transport

		END_IF

	END_IF

END_FUNCTION
```

#### fHermesChkParamSOT.st
```iecst
(* Hermes Checking Parameter Stop Transport *)
FUNCTION fHermesChkParamSOT

	fHermesChkParamSOT	:= 0;

	IF fHermesChkParamSOT = 0 THEN

		IF tyStopTransport.tyAvl.bTransferState = FALSE THEN

			fHermesChkParamSOT	:= 2742;	//TransferState Missing While Checking Stop Transport

		END_IF

	END_IF

	IF fHermesChkParamSOT = 0 THEN

		IF tyStopTransport.tyAvl.bBoardId = FALSE THEN

			fHermesChkParamSOT	:= 2743;	//BoardId Missing While Checking Stop Transport

		END_IF

	END_IF

END_FUNCTION
```

#### fHermesChkParamTF.st
```iecst
(* Hermes Checking Parameter Transport Finished *)
FUNCTION fHermesChkParamTF

	fHermesChkParamTF	:= 0;

	IF fHermesChkParamTF = 0 THEN

		IF tyTransportFinished.tyAvl.bTransferState = FALSE THEN

			fHermesChkParamTF	:= 2744;	//TransferState Missing While Checking Transport Finished

		END_IF

	END_IF

	IF fHermesChkParamTF = 0 THEN

		IF tyTransportFinished.tyAvl.bBoardId = FALSE THEN

			fHermesChkParamTF	:= 2745;	//BoardId Missing While Checking Transport Finished

		END_IF

	END_IF

END_FUNCTION
```

#### fHermesChkParamSC.st
```iecst
(* Hermes Checking Parameter Set Configuration *)
FUNCTION fHermesChkParamSC

	fHermesChkParamSC	:= 0;

	IF fHermesChkParamSC = 0 THEN

		IF tySetConfiguration.tyAvl.bMachineId = TRUE THEN

			IF tySetConfiguration.tyData.sMachineId <> sMachineId THEN

				fHermesChkParamSC	:= 2746;	//MachineId Mismatch While Checking Set Configuration

			END_IF

		ELSE

			fHermesChkParamSC	:= 2747;	//MachineId Missing While Checking Set Configuration

		END_IF

	END_IF

	IF fHermesChkParamSC = 0 THEN

		FOR i := 0 TO tySetConfiguration.tyAvl.iUpstreamConfigurations DO

			IF tySetConfiguration.tyAvl.a_tyUpstreamConfigurations[i].bUpstreamLaneId = TRUE THEN

				IF tySetConfiguration.tyData.a_tyUpstreamConfigurations[i].iUpstreamLaneId <= 0 THEN

					fHermesChkParamSC	:= 2748;	//UpstreamLaneId Out Of Range While Checking Set Configuration
					EXIT;

				END_IF

			ELSE

				fHermesChkParamSC	:= 2749;	//UpstreamLaneId Missing While Checking Set Configuration
				EXIT;

			END_IF

			IF tySetConfiguration.tyAvl.a_tyUpstreamConfigurations[i].bHostAddress = TRUE THEN

				IF (fIPValid(tySetConfiguration.tyData.a_tyUpstreamConfigurations[i].sHostAddress , ADR(a_iIPPart))) = FALSE THEN

					fHermesChkParamSC	:= 2750;	//HostAddress Invalid While Checking Set Configuration
					EXIT;

				END_IF

			ELSE

				fHermesChkParamSC	:= 2751;	//HostAddress Missing While Checking Set Configuration
				EXIT;

			END_IF

		END_FOR

	END_IF

	IF fHermesChkParamSC = 0 THEN

		FOR i := 0 TO tySetConfiguration.tyAvl.iDownstreamConfigurations DO

			IF tySetConfiguration.tyAvl.a_tyDownstreamConfigurations[i].bDownstreamLaneId = TRUE THEN

				IF tySetConfiguration.tyData.a_tyDownstreamConfigurations[i].iDownstreamLaneId <= 0 THEN

					fHermesChkParamSC	:= 2752;	//DownstreamLaneId Out Of Range While Checking Set Configuration
					EXIT;

				END_IF

			ELSE

				fHermesChkParamSC	:= 2753;	//DownstreamLaneId Missing While Checking Set Configuration
				EXIT;

			END_IF

			IF tySetConfiguration.tyAvl.a_tyDownstreamConfigurations[i].bClientAddress = TRUE THEN

				IF (fIPValid(tySetConfiguration.tyData.a_tyDownstreamConfigurations[i].sClientAddress , ADR(a_iIPPart))) = FALSE THEN

					fHermesChkParamSC	:= 2754;	//ClientAddress Invalid While Checking Set Configuration
					EXIT;

				END_IF

			END_IF

		END_FOR

	END_IF

END_FUNCTION
```

#### fHermesChkParamCC.st
```iecst
(* Hermes Checking Parameter Current Configuration *)
FUNCTION fHermesChkParamCC

	fHermesChkParamCC	:= 0;

	IF fHermesChkParamCC = 0 THEN

		IF tyCurrentConfiguration.tyAvl.bMachineId = TRUE THEN

			IF tyCurrentConfiguration.tyData.sMachineId <> sMachineId THEN

				fHermesChkParamCC	:= 2755;	//MachineId Mismatch While Checking Current Configuration

			END_IF

		ELSE

			fHermesChkParamCC	:= 2756;	//MachineId Missing While Checking Current Configuration

		END_IF

	END_IF

	IF fHermesChkParamCC = 0 THEN

		FOR i := 0 TO tyCurrentConfiguration.tyAvl.iUpstreamConfigurations DO

			IF tyCurrentConfiguration.tyAvl.a_tyUpstreamConfigurations[i].bUpstreamLaneId = TRUE THEN

				IF tyCurrentConfiguration.tyData.a_tyUpstreamConfigurations[i].iUpstreamLaneId <= 0 THEN

					fHermesChkParamCC	:= 2757;	//UpstreamLaneId Out Of Range While Checking Current Configuration
					EXIT;

				END_IF

			ELSE

				fHermesChkParamCC	:= 2758;	//UpstreamLaneId Missing While Checking Current Configuration
				EXIT;

			END_IF

			IF tyCurrentConfiguration.tyAvl.a_tyUpstreamConfigurations[i].bHostAddress = TRUE THEN

				IF (fIPValid(tyCurrentConfiguration.tyData.a_tyUpstreamConfigurations[i].sHostAddress , ADR(a_iIPPart))) = FALSE THEN

					fHermesChkParamCC	:= 2759;	//HostAddress Invalid While Checking Current Configuration
					EXIT;

				END_IF

			ELSE

				fHermesChkParamCC	:= 2760;	//HostAddress Missing While Checking Current Configuration
				EXIT;

			END_IF

		END_FOR

	END_IF

	IF fHermesChkParamCC = 0 THEN

		FOR i := 0 TO tyCurrentConfiguration.tyAvl.iDownstreamConfigurations DO

			IF tyCurrentConfiguration.tyAvl.a_tyDownstreamConfigurations[i].bDownstreamLaneId = TRUE THEN

				IF tyCurrentConfiguration.tyData.a_tyDownstreamConfigurations[i].iDownstreamLaneId <= 0 THEN

					fHermesChkParamCC	:= 2761;	//DownstreamLaneId Out Of Range While Checking Current Configuration
					EXIT;

				END_IF

			ELSE

				fHermesChkParamCC	:= 2762;	//DownstreamLaneId Missing While Checking Current Configuration
				EXIT;

			END_IF

			IF tyCurrentConfiguration.tyAvl.a_tyDownstreamConfigurations[i].bClientAddress = TRUE THEN

				IF (fIPValid(tyCurrentConfiguration.tyData.a_tyDownstreamConfigurations[i].sClientAddress , ADR(a_iIPPart))) = FALSE THEN

					fHermesChkParamCC	:= 2763;	//ClientAddress Invalid While Checking Current Configuration
					EXIT;

				END_IF

			END_IF

		END_FOR

	END_IF

END_FUNCTION
```

#### fHermesChkParamBF.st
```iecst
(* Hermes Checking Parameter Board Forecast *)
FUNCTION fHermesChkParamBF

	fHermesChkParamBF	:= 0;

	IF fHermesChkParamBF = 0 THEN

		IF tyBoardForecast.tyAvl.bFailedBoard = FALSE THEN

			fHermesChkParamBF	:= 2764;	//FailedBoard Missing While Checking Board Forecast

		END_IF

	END_IF

	IF fHermesChkParamBF = 0 THEN

		IF tyBoardForecast.tyAvl.bFlippedBoard = FALSE THEN

			fHermesChkParamBF	:= 2765;	//FlippedBoard Missing While Checking Board Forecast

		END_IF

	END_IF

END_FUNCTION
```

#### fHermesChkParamQBI.st
```iecst
(* Hermes Checking Parameter Query Board Info *)
FUNCTION fHermesChkParamQBI

	fHermesChkParamQBI	:= 0;

	IF fHermesChkParamQBI = 0 THEN

		IF tyQueryBoardInfo.tyAvl.bTopBarcode = FALSE AND tyQueryBoardInfo.tyAvl.bBottomBarcode = FALSE THEN

			fHermesChkParamQBI	:= 2766;	//Barcode Missing While Checking Query Board Info

		END_IF

	END_IF

END_FUNCTION
```

#### fHermesChkParamSBIQBI.st
```iecst
(* Hermes Checking Parameter SendBoardInfo & QueryBoardInfo *)
FUNCTION fHermesChkParamSBIQBI

	fHermesChkParamSBIQBI	:= 0;

	IF tyQueryBoardInfo.tyAvl.bTopBarcode = TRUE THEN

		IF tySendBoardInfo.tyAvl.bTopBarcode = TRUE THEN

			IF tySendBoardInfo.tyData.sTopBarcode <> tyQueryBoardInfo.tyData.sTopBarcode THEN

			fHermesChkParamSBIQBI	:= 2769;	//Top Barcode Mismatch While Checking SendBoardInfo & QueryBoardInfo

			END_IF
		ELSE
			fHermesChkParamSBIQBI	:= 2770;	//Top Barcode Missing While Checking SendBoardInfo & QueryBoardInfo
		END_IF
	ELSE
		IF tySendBoardInfo.tyAvl.bTopBarcode = TRUE THEN

			fHermesChkParamSBIQBI	:= 2769;	//Bottom Barcode Mismatch While Checking SendBoardInfo & QueryBoardInfo
		END_IF
	END_IF

	IF tyQueryBoardInfo.tyAvl.bBottomBarcode = TRUE THEN

		IF tySendBoardInfo.tyAvl.bBottomBarcode = TRUE THEN

			IF tySendBoardInfo.tyData.sBottomBarcode <> tyQueryBoardInfo.tyData.sBottomBarcode THEN

				fHermesChkParamSBIQBI	:= 2771;	//Bottom Barcode Mismatch While Checking SendBoardInfo & QueryBoardInfo

			END_IF
		ELSE
			fHermesChkParamSBIQBI	:= 2772;	//Bottom Barcode Missing While Checking SendBoardInfo & QueryBoardInfo
		END_IF

	ELSE
		IF tySendBoardInfo.tyAvl.bBottomBarcode = TRUE THEN

			fHermesChkParamSBIQBI	:= 2771;	//Bottom Barcode Mismatch While Checking SendBoardInfo & QueryBoardInfo
		END_IF
	END_IF

END_FUNCTION
```

#### fHermesChkParamSWQW.st
```iecst
(* Hermes Checking Parameter SendWorkOrderId & QueryWorkOrderId *)
FUNCTION fHermesChkParamSWQW

	fHermesChkParamSWQW	:= 0;

	IF tySendWorkOrderInfo.tyAvl.bQueryId = TRUE AND tyQueryWorkOrderInfo.tyAvl.bQueryId = TRUE THEN

		IF tySendWorkOrderInfo.tyData.sQueryId <> tyQueryWorkOrderInfo.tyData.sQueryId THEN

			fHermesChkParamSWQW	:= 2767;	//QueryId Mismatch While Checking SendWorkOrderId & QueryWorkOrderId

		END_IF

	ELSE

		fHermesChkParamSWQW	:= 2768;	//QueryId Missing While Checking SendWorkOrderId & QueryWorkOrderId

	END_IF

END_FUNCTION
```

#### fHermesNotificationRstConn.st
```iecst
(* Hermes Notification Reset Connection *)
FUNCTION fHermesNotificationRstConn

	IF tyNotification.tyData.eSeverity = HermesSeverityFatalError THEN

		fHermesNotificationRstConn	:= TRUE;

	ELSE

		fHermesNotificationRstConn	:= FALSE;

	END_IF

END_FUNCTION
```

#### fHermesNotificationRstState.st
```iecst
(* Hermes Notification Reset State *)
FUNCTION fHermesNotificationRstState

	IF tyNotification.tyData.eSeverity = HermesSeverityFatalError THEN

		fHermesNotificationRstState	:= TRUE;

	ELSIF tyNotification.tyData.eSeverity = HermesSeverityError THEN

		fHermesNotificationRstState	:= TRUE;

	ELSE

		fHermesNotificationRstState	:= FALSE;

	END_IF

END_FUNCTION
```

#### fbHermesCheckAlive.st
```iecst
(* Hermes Check Alive *)
FUNCTION_BLOCK fbHermesCheckAlive

	IF (bEn = TRUE) AND (udiStatus >= 65534) THEN

		udiStatus	:= 65535;

		//Send Check Alive
		fbSendTm(IN := TRUE , PT := tSendTm);
		IF fbSendTm.Q = TRUE THEN
			fbSendTm(IN := FALSE);

			bDataSend	:= TRUE;
			memset(ADR(tyDataSend) , 0 , SIZEOF(tyDataSend));

		ELSE
			bDataSend	:= FALSE;
		END_IF

		//Wait Check Alive
		fbRcvTO(IN := NOT EDGEPOS(bDataRcv) , PT := tRcvTimeOut);
		IF fbRcvTO.Q = TRUE THEN
			udiStatus	:= 2767;	//Waiting Check Alive Time Out
		END_IF

	ELSIF (bEn = FALSE) AND (udiStatus <> 65534) THEN

		udiStatus	:= 65534;

		bDataSend	:= FALSE;
		memset(ADR(tyDataSend) , 0 , SIZEOF(tyDataSend));

		fbSendTm(IN := FALSE);
		fbRcvTO(IN := FALSE);

	END_IF

END_FUNCTION_BLOCK
```

#### fbHermesCheckAliveSendPing.st
```iecst
(* Hermes Check Alive Send Ping Wait Pong *)
FUNCTION_BLOCK fbHermesCheckAliveSendPing

	IF (bEn = TRUE) AND (udiStatus >= 65534) THEN

		udiStatus	:= 65535;

		//Send Check Alive
		fbSendTm(IN := TRUE , PT := tSendTm);
		IF fbSendTm.Q = TRUE THEN
			fbSendTm(IN := FALSE);

			bDataSend				:= TRUE;
			tyDataSend.tyAvl.bType	:= TRUE;
			tyDataSend.tyAvl.bId	:= TRUE;
			tyDataSend.tyData.eType	:= HermesCheckAliveTypePing;
			fHermesGetTimestamp(ADR(tyDataSend.tyData.sId) , tyDTStructure);

		ELSE
			bDataSend	:= FALSE;
		END_IF

		//Wait Check Alive
		fbRcvTO(IN := NOT EDGEPOS(bDataRcv) , PT := tRcvTimeOut);
		IF fbRcvTO.Q = TRUE THEN
			udiStatus	:= 2768;	//Waiting Check Alive Time Out
		END_IF

		IF EDGEPOS(bDataRcv) THEN
			IF tyDataRcv.tyData.sId <> tyDataSend.tyData.sId THEN
				udiStatus	:= 2769;	//Check Alive Id Mismatch
			END_IF
		END_IF

	ELSIF (bEn = FALSE) AND (udiStatus <> 65534) THEN

		udiStatus	:= 65534;

		bDataSend	:= FALSE;
		memset(ADR(tyDataSend) , 0 , SIZEOF(tyDataSend));

		fbSendTm(IN := FALSE);
		fbRcvTO(IN := FALSE);

	END_IF

END_FUNCTION_BLOCK
```

#### fbHermesCheckAliveRcvPing.st
```iecst
(* Hermes Check Alive Receive Ping Send Pong *)
FUNCTION_BLOCK fbHermesCheckAliveRcvPing

	IF (bEn = TRUE) AND (udiStatus >= 65534) THEN

		udiStatus	:= 65535;

		IF EDGEPOS(bDataRcv) THEN

			bDataSend				:= TRUE;
			tyDataSend.tyAvl.bType	:= TRUE;
			tyDataSend.tyAvl.bId	:= TRUE;
			tyDataSend.tyData.eType	:= HermesCheckAliveTypePong;
			tyDataSend.tyData.sId	:= tyDataRcv.tyData.sId;

		ELSE

			bDataSend	:= FALSE;
			memset(ADR(tyDataSend) , 0 , SIZEOF(tyDataSend));

		END_IF

	ELSIF (bEn = FALSE) AND (udiStatus <> 65534) THEN

		udiStatus	:= 65534;

		bDataSend	:= FALSE;
		memset(ADR(tyDataSend) , 0 , SIZEOF(tyDataSend));

	END_IF

END_FUNCTION_BLOCK
```

#### fHermesIllegalMsgUS.st
```iecst
(* Hermes Illegal Message - Upstream *)
FUNCTION fHermesIllegalMsgUS

	CASE eState OF

		HermesStateNotConnected:			fHermesIllegalMsgUS	:= fHermesIllegalMsgNotConnectedUS(tyMsgType); //2770 - 2778
		HermesStateServiceDescription:		fHermesIllegalMsgUS	:= fHermesIllegalMsgSrvcDescripUS(tyMsgType); //2779 - 2786
		HermesStateNotAvailableNotReady:	fHermesIllegalMsgUS	:= fHermesIllegalMsgNotAvlNotRdyUS(tyMsgType); //2787 - 2793
		HermesStateBoardAvailable:			fHermesIllegalMsgUS	:= fHermesIllegalMsgBrdAvlUS(tyMsgType); //2794 - 2801
		HermesStateMachineReady:			fHermesIllegalMsgUS	:= fHermesIllegalMsgMcRdyUS(tyMsgType); //2802 - 2808
		HermesStateAvailableAndReady:		fHermesIllegalMsgUS	:= fHermesIllegalMsgAvlAndRdyUS(tyMsgType); //2809 - 2816
		HermesStateTransporting:			fHermesIllegalMsgUS	:= fHermesIllegalMsgTransportingUS(tyMsgType , bBoardAvailable); //2817-2823
		HermesStateTransportFinished:		fHermesIllegalMsgUS	:= fHermesIllegalMsgTransportFiniUS(tyMsgType); //2824 - 2832
		HermesStateTransportStopped:		fHermesIllegalMsgUS	:= fHermesIllegalMsgTransportStopUS(tyMsgType , bBoardAvailable); //2833 - 2839

	END_CASE

END_FUNCTION
```

#### fHermesIllegalMsgDS.st
```iecst
(* Hermes Illegal Message - Downstream *)
FUNCTION fHermesIllegalMsgDS

	CASE eState OF

		HermesStateNotConnected:			fHermesIllegalMsgDS	:= fHermesIllegalMsgNotConnectedDS(tyMsgType); //2840 - 2847
		HermesStateServiceDescription:		fHermesIllegalMsgDS	:= fHermesIllegalMsgSrvcDescripDS(tyMsgType); //2848 - 2856
		HermesStateNotAvailableNotReady:	fHermesIllegalMsgDS	:= fHermesIllegalMsgNotAvlNotRdyDS(tyMsgType); //2857 - 2864
		HermesStateBoardAvailable:			fHermesIllegalMsgDS	:= fHermesIllegalMsgBrdAvlDS(tyMsgType);  //2865 - 2872
		HermesStateMachineReady:			fHermesIllegalMsgDS	:= fHermesIllegalMsgMcRdyDS(tyMsgType); //2873 - 2879
		HermesStateAvailableAndReady:		fHermesIllegalMsgDS	:= fHermesIllegalMsgAvlAndRdyDS(tyMsgType); //2880 - 2886
		HermesStateTransporting:			fHermesIllegalMsgDS	:= fHermesIllegalMsgTransportingDS(tyMsgType); //2887 - 2894
		HermesStateTransportStopped:		fHermesIllegalMsgDS	:= fHermesIllegalMsgTransportStopDS(tyMsgType); //2903 - 2911
		HermesStateTransportFinished:		fHermesIllegalMsgDS	:= fHermesIllegalMsgTransportFiniDS(tyMsgType); //2895 - 2902

	END_CASE

END_FUNCTION
```

#### fHermesIllegalMsgRmt.st
```iecst
(* Hermes Illegal Message - Remote Configuration *)
FUNCTION fHermesIllegalMsgRmt //2925 - 2939

	IF tyMsgType.bCheckAlive = TRUE THEN

		fHermesIllegalMsgRmt	:= 2925;	//Receive Check Alive While In Remote Configuration

	ELSIF tyMsgType.bCheckAlivePing = TRUE THEN

		fHermesIllegalMsgRmt	:= 2926;	//Receive Check Alive Ping While In Remote Configuration

	ELSIF tyMsgType.bCheckAlivePong = TRUE THEN

		fHermesIllegalMsgRmt	:= 2927;	//Receive Check Alive Pong While In Remote Configuration

	ELSIF tyMsgType.bServiceDescription = TRUE THEN

		fHermesIllegalMsgRmt	:= 2928;	//Receive ServiceDescription While In Remote Configuration

	ELSIF tyMsgType.bBoardAvailable = TRUE THEN

		fHermesIllegalMsgRmt	:= 2929;	//Receive BoardAvailable While In Remote Configuration

	ELSIF tyMsgType.bRevokeBoardAvailable = TRUE THEN

		fHermesIllegalMsgRmt	:= 2930;	//Receive RevokeBoardAvailable While In Remote Configuration

	ELSIF tyMsgType.bMachineReady = TRUE THEN

		fHermesIllegalMsgRmt	:= 2931;	//Receive MachineReady While In Remote Configuration

	ELSIF tyMsgType.bRevokeMachineReady = TRUE THEN

		fHermesIllegalMsgRmt	:= 2932;	//Receive RevokeMachineReady While In Remote Configuration

	ELSIF tyMsgType.bStartTransport = TRUE THEN

		fHermesIllegalMsgRmt	:= 2933;	//Receive StartTransport While In Remote Configuration

	ELSIF tyMsgType.bStopTransport = TRUE THEN

		fHermesIllegalMsgRmt	:= 2934;	//Receive StopTransport While In Remote Configuration

	ELSIF tyMsgType.bTransportFinished = TRUE THEN

		fHermesIllegalMsgRmt	:= 2935;	//Receive TransportFinished While In Remote Configuration

	ELSIF tyMsgType.bCurrentConfiguration = TRUE THEN

		fHermesIllegalMsgRmt	:= 2936;	//Receive CurrentConfiguration While In Remote Configuration

	ELSIF tyMsgType.bBoardForecast = TRUE THEN

		fHermesIllegalMsgRmt	:= 2937;	//Receive BoardForecast While In Remote Configuration

	ELSIF tyMsgType.bQueryBoardInfo = TRUE THEN

		fHermesIllegalMsgRmt	:= 2938;	//Receive QueryBoardInfo While In Remote Configuration

	ELSIF tyMsgType.bSendBoardInfo = TRUE THEN

		fHermesIllegalMsgRmt	:= 2939;	//Receive SendBoardInfo While In Remote Configuration

	ELSE

		fHermesIllegalMsgRmt	:= 0;

	END_IF

END_FUNCTION
```

#### fHermesIllegalMsgSvy.st
```iecst
(* Hermes Illegal Message - Supervisory *)
FUNCTION fHermesIllegalMsgSvy

	CASE eState OF

		HermesStateNotConnected:			fHermesIllegalMsgSvy	:= fHermesIllegalMsgNotConnectedSvy(tyMsgType); //2940 - 2946, 4 standby until 2950
		HermesStateSServiceDescription:  	fHermesIllegalMsgSvy	:= fHermesIllegalMsgSrvcDescripSvy(tyMsgType); //2951 - 2958, 4 standby until 2962
		HermesStateConnected:               fHermesIllegalMsgSvy	:= fHermesIllegalMsgConnectedSvy(tyMsgType); //2963 - 2967, 4 standby until 2971

	END_CASE

END_FUNCTION
```

#### fHermesIllegalMsgNotConnectedUS.st
```iecst
(* Hermes Illegal Message - Not Connected For Upstream *)
FUNCTION fHermesIllegalMsgNotConnectedUS

	IF tyMsgType.bServiceDescription = TRUE THEN

		fHermesIllegalMsgNotConnectedUS	:= 2770;	//Receive ServiceDescription While Upstream In Not Connected State

	ELSIF tyMsgType.bBoardAvailable = TRUE THEN

		fHermesIllegalMsgNotConnectedUS	:= 2771;	//Receive BoardAvailable While Upstream In Not Connected State

	ELSIF tyMsgType.bRevokeBoardAvailable = TRUE THEN

		fHermesIllegalMsgNotConnectedUS	:= 2772;	//Receive RevokeBoardAvailable While Upstream In Not Connected State

	ELSIF tyMsgType.bMachineReady = TRUE THEN

		fHermesIllegalMsgNotConnectedUS	:= 2773;	//Receive MachineReady While Upstream In Not Connected State

	ELSIF tyMsgType.bRevokeMachineReady = TRUE THEN

		fHermesIllegalMsgNotConnectedUS	:= 2774;	//Receive RevokeMachineReady While Upstream In Not Connected State

	ELSIF tyMsgType.bStartTransport = TRUE THEN

		fHermesIllegalMsgNotConnectedUS	:= 2775;	//Receive StartTransport While Upstream In Not Connected State

	ELSIF tyMsgType.bStopTransport = TRUE THEN

		fHermesIllegalMsgNotConnectedUS	:= 2776;	//Receive StopTransport While Upstream In Not Connected State

	ELSIF tyMsgType.bTransportFinished = TRUE THEN

		fHermesIllegalMsgNotConnectedUS	:= 2777;	//Receive TransportFinished While Upstream In Not Connected State

	ELSIF tyMsgType.bBoardForecast = TRUE THEN

		fHermesIllegalMsgNotConnectedUS	:= 2778;	//Receive BoardForecast While Upstream In Not Connected State

	ELSE

		fHermesIllegalMsgNotConnectedUS	:= 0;

	END_IF

END_FUNCTION
```

#### fHermesIllegalMsgSrvcDescripUS.st
```iecst
(* Hermes Illegal Message - Service Description For Upstream *)
FUNCTION fHermesIllegalMsgSrvcDescripUS

//	IF tyMsgType.bBoardAvailable = TRUE THEN //Commented due to ASM can send B.A message immediately (0.01 sec) after send us Service description before our machine can react and change Hermes eState from HermesStateServiceDescription to HermesStateNotAvailableNotReady
//
//		fHermesIllegalMsgSrvcDescripUS	:= 2779;	//Receive BoardAvailable While Upstream In Service Description State

	IF tyMsgType.bRevokeBoardAvailable = TRUE THEN

		fHermesIllegalMsgSrvcDescripUS	:= 2780;	//Receive RevokeBoardAvailable While Upstream In Service Description State

	ELSIF tyMsgType.bMachineReady = TRUE THEN

		fHermesIllegalMsgSrvcDescripUS	:= 2781;	//Receive MachineReady While Upstream In Service Description State

	ELSIF tyMsgType.bRevokeMachineReady = TRUE THEN

		fHermesIllegalMsgSrvcDescripUS	:= 2782;	//Receive RevokeMachineReady While Upstream In Service Description State

	ELSIF tyMsgType.bStartTransport = TRUE THEN

		fHermesIllegalMsgSrvcDescripUS	:= 2783;	//Receive StartTransport While Upstream In Service Description State

	ELSIF tyMsgType.bStopTransport = TRUE THEN

		fHermesIllegalMsgSrvcDescripUS	:= 2784;	//Receive StopTransport While Upstream In Service Description State

	ELSIF tyMsgType.bTransportFinished = TRUE THEN

		fHermesIllegalMsgSrvcDescripUS	:= 2785;	//Receive TransportFinished While Upstream In Service Description State

//	ELSIF tyMsgType.bBoardForecast = TRUE THEN //Commented due to ASM can send B.F message immediately (0.01 sec) after send us Service description before our machine can react and change Hermes eState from HermesStateServiceDescription to HermesStateNotAvailableNotReady
//
//		fHermesIllegalMsgSrvcDescripUS	:= 2786;	//Receive BoardForecast While Upstream In Service Description State

	ELSE

		fHermesIllegalMsgSrvcDescripUS	:= 0;

	END_IF

END_FUNCTION
```

#### fHermesIllegalMsgNotAvlNotRdyUS.st
```iecst
(* Hermes Illegal Message - Not Available Not Ready For Upstream *)
FUNCTION fHermesIllegalMsgNotAvlNotRdyUS

	IF tyMsgType.bServiceDescription = TRUE THEN

		fHermesIllegalMsgNotAvlNotRdyUS	:= 2787;	//Receive ServiceDescription While Upstream In Not Available Not Ready State

	ELSIF tyMsgType.bRevokeBoardAvailable = TRUE THEN

		fHermesIllegalMsgNotAvlNotRdyUS	:= 2788;	//Receive RevokeBoardAvailable While Upstream In Not Available Not Ready State

	ELSIF tyMsgType.bMachineReady = TRUE THEN

		fHermesIllegalMsgNotAvlNotRdyUS	:= 2789;	//Receive MachineReady While Upstream In Not Available Not Ready State

	ELSIF tyMsgType.bRevokeMachineReady = TRUE THEN

		fHermesIllegalMsgNotAvlNotRdyUS	:= 2790;	//Receive RevokeMachineReady While Upstream In Not Available Not Ready State

	ELSIF tyMsgType.bStartTransport = TRUE THEN

		fHermesIllegalMsgNotAvlNotRdyUS	:= 2791;	//Receive StartTransport While Upstream In Not Available Not Ready State

	ELSIF tyMsgType.bStopTransport = TRUE THEN

		fHermesIllegalMsgNotAvlNotRdyUS	:= 2792;	//Receive StopTransport While Upstream In Not Available Not Ready State

	ELSIF tyMsgType.bTransportFinished = TRUE THEN

		fHermesIllegalMsgNotAvlNotRdyUS	:= 2793;	//Receive TransportFinished While Upstream In Not Available Not Ready State

	ELSE

		fHermesIllegalMsgNotAvlNotRdyUS	:= 0;

	END_IF

END_FUNCTION
```

#### fHermesIllegalMsgBrdAvlUS.st
```iecst
(* Hermes Illegal Message - Board Available For Upstream *)
FUNCTION fHermesIllegalMsgBrdAvlUS

	IF tyMsgType.bServiceDescription = TRUE THEN

		fHermesIllegalMsgBrdAvlUS	:= 2794;	//Receive ServiceDescription While Upstream In Board Available State

	ELSIF tyMsgType.bBoardAvailable = TRUE THEN

		fHermesIllegalMsgBrdAvlUS	:= 2795;	//Receive BoardAvailable While Upstream In Board Available State

	ELSIF tyMsgType.bMachineReady = TRUE THEN

		fHermesIllegalMsgBrdAvlUS	:= 2796;	//Receive MachineReady While Upstream In Board Available State

	ELSIF tyMsgType.bRevokeMachineReady = TRUE THEN

		fHermesIllegalMsgBrdAvlUS	:= 2797;	//Receive RevokeMachineReady While Upstream In Board Available State

	ELSIF tyMsgType.bStartTransport = TRUE THEN

		fHermesIllegalMsgBrdAvlUS	:= 2798;	//Receive StartTransport While Upstream In Board Available State

	ELSIF tyMsgType.bStopTransport = TRUE THEN

		fHermesIllegalMsgBrdAvlUS	:= 2799;	//Receive StopTransport While Upstream In Board Available State

	ELSIF tyMsgType.bTransportFinished = TRUE THEN

		fHermesIllegalMsgBrdAvlUS	:= 2800;	//Receive TransportFinished While Upstream In Board Available State

//	ELSIF tyMsgType.bBoardForecast = TRUE THEN
//
//		fHermesIllegalMsgBrdAvlUS	:= 2801;	//Receive BoardForecast While Upstream In Board Available State

	ELSE

		fHermesIllegalMsgBrdAvlUS	:= 0;

	END_IF

END_FUNCTION
```

#### fHermesIllegalMsgMcRdyUS.st
```iecst
(* Hermes Illegal Message - Machine Ready For Upstream *)
FUNCTION fHermesIllegalMsgMcRdyUS

	IF tyMsgType.bServiceDescription = TRUE THEN

		fHermesIllegalMsgMcRdyUS	:= 2802;	//Receive ServiceDescription While Upstream In Machine Ready State

	ELSIF tyMsgType.bRevokeBoardAvailable = TRUE THEN

		fHermesIllegalMsgMcRdyUS	:= 2803;	//Receive RevokeBoardAvailable While Upstream In Machine Ready State

	ELSIF tyMsgType.bMachineReady = TRUE THEN

		fHermesIllegalMsgMcRdyUS	:= 2804;	//Receive MachineReady While Upstream In Machine Ready State

	ELSIF tyMsgType.bRevokeMachineReady = TRUE THEN

		fHermesIllegalMsgMcRdyUS	:= 2805;	//Receive RevokeMachineReady While Upstream In Machine Ready State

	ELSIF tyMsgType.bStartTransport = TRUE THEN

		fHermesIllegalMsgMcRdyUS	:= 2806;	//Receive StartTransport While Upstream In Machine Ready State

	ELSIF tyMsgType.bStopTransport = TRUE THEN

		fHermesIllegalMsgMcRdyUS	:= 2807;	//Receive StopTransport While Upstream In Machine Ready State

	ELSIF tyMsgType.bTransportFinished = TRUE THEN

		fHermesIllegalMsgMcRdyUS	:= 2808;	//Receive TransportFinished While Upstream In Machine Ready State

	ELSE

		fHermesIllegalMsgMcRdyUS	:= 0;

	END_IF

END_FUNCTION
```

#### fHermesIllegalMsgAvlAndRdyUS.st
```iecst
(* Hermes Illegal Message - Available And Ready For Upstream *)
FUNCTION fHermesIllegalMsgAvlAndRdyUS

	IF tyMsgType.bServiceDescription = TRUE THEN

		fHermesIllegalMsgAvlAndRdyUS	:= 2809;	//Receive ServiceDescription While Upstream In Available And Ready State

	ELSIF tyMsgType.bBoardAvailable = TRUE THEN

		fHermesIllegalMsgAvlAndRdyUS	:= 2810;	//Receive BoardAvailable While Upstream In Available And Ready State

	ELSIF tyMsgType.bMachineReady = TRUE THEN

		fHermesIllegalMsgAvlAndRdyUS	:= 2811;	//Receive MachineReady While Upstream In Available And Ready State

	ELSIF tyMsgType.bRevokeMachineReady = TRUE THEN

		fHermesIllegalMsgAvlAndRdyUS	:= 2812;	//Receive RevokeMachineReady While Upstream In Available And Ready State

	ELSIF tyMsgType.bStartTransport = TRUE THEN

		fHermesIllegalMsgAvlAndRdyUS	:= 2813;	//Receive StartTransport While Upstream In Available And Ready State

	ELSIF tyMsgType.bStopTransport = TRUE THEN

		fHermesIllegalMsgAvlAndRdyUS	:= 2814;	//Receive StopTransport While Upstream In Available And Ready State

	ELSIF tyMsgType.bTransportFinished = TRUE THEN

		fHermesIllegalMsgAvlAndRdyUS	:= 2815;	//Receive TransportFinished While Upstream In Available And Ready State

//	ELSIF tyMsgType.bBoardForecast = TRUE THEN
//
//		fHermesIllegalMsgAvlAndRdyUS	:= 2816;	//Receive BoardForecast While Upstream In Available And Ready State

	ELSE

		fHermesIllegalMsgAvlAndRdyUS	:= 0;

	END_IF

END_FUNCTION
```

#### fHermesIllegalMsgTransportingUS.st
```iecst
(* Hermes Illegal Message - Transporting For Upstream *)
FUNCTION fHermesIllegalMsgTransportingUS

	IF tyMsgType.bServiceDescription = TRUE THEN

		fHermesIllegalMsgTransportingUS	:= 2817;	//Receive ServiceDescription While Upstream In Transporting State

	ELSIF tyMsgType.bBoardAvailable = TRUE AND bBoardAvailable = TRUE THEN

		fHermesIllegalMsgTransportingUS	:= 2818;	//Receive Twice Board Available While Upstream In Transporting State

	ELSIF tyMsgType.bRevokeBoardAvailable = TRUE AND bBoardAvailable = FALSE THEN

		fHermesIllegalMsgTransportingUS	:= 2819;	//Receive RevokeBoardAvailable Without BoardAvailable While Upstream In Transporting State

	ELSIF tyMsgType.bMachineReady = TRUE THEN

		fHermesIllegalMsgTransportingUS	:= 2820;	//Receive MachineReady While Upstream In Transporting State

	ELSIF tyMsgType.bRevokeMachineReady = TRUE THEN

		fHermesIllegalMsgTransportingUS	:= 2821;	//Receive RevokeMachineReady While Upstream In Transporting State

	ELSIF tyMsgType.bStartTransport = TRUE THEN

		fHermesIllegalMsgTransportingUS	:= 2822;	//Receive StartTransport While Upstream In Transporting State

	ELSIF tyMsgType.bStopTransport = TRUE THEN

		fHermesIllegalMsgTransportingUS	:= 2823;	//Receive StopTransport While Upstream In Transporting State

	ELSE

		fHermesIllegalMsgTransportingUS	:= 0;

	END_IF

END_FUNCTION
```

#### fHermesIllegalMsgTransportFiniUS.st
```iecst
(* Hermes Illegal Message - Transport Finished For Upstream *)
FUNCTION fHermesIllegalMsgTransportFiniUS

	IF tyMsgType.bServiceDescription = TRUE THEN

		fHermesIllegalMsgTransportFiniUS	:= 2824;	//Receive ServiceDescription While Upstream In Transport Finished State

	ELSIF tyMsgType.bBoardAvailable = TRUE THEN

		fHermesIllegalMsgTransportFiniUS	:= 2825;	//Receive BoardAvailable While Upstream In Transport Finished State

	ELSIF tyMsgType.bRevokeBoardAvailable = TRUE THEN

		fHermesIllegalMsgTransportFiniUS	:= 2826;	//Receive RevokeBoardAvailable While UpstreamWhile Upstream In Transport Finished State

	ELSIF tyMsgType.bMachineReady = TRUE THEN

		fHermesIllegalMsgTransportFiniUS	:= 2827;	//Receive MachineReady While Upstream In Transport Finished State

	ELSIF tyMsgType.bRevokeMachineReady = TRUE THEN

		fHermesIllegalMsgTransportFiniUS	:= 2828;	//Receive RevokeMachineReady While Upstream In Transport Finished State

	ELSIF tyMsgType.bStartTransport = TRUE THEN

		fHermesIllegalMsgTransportFiniUS	:= 2829;	//Receive StartTransport While Upstream In Transport Finished State

	ELSIF tyMsgType.bTransportFinished = TRUE THEN

		fHermesIllegalMsgTransportFiniUS	:= 2830;	//Receive TransportFinished While Upstream In Transport Finished State

	ELSIF tyMsgType.bStopTransport = TRUE THEN

		fHermesIllegalMsgTransportFiniUS	:= 2831;	//Receive StopTransport While Upstream In Transport Finished State

//	ELSIF tyMsgType.bBoardForecast = TRUE THEN
//
//		fHermesIllegalMsgTransportFiniUS	:= 2832;	//Receive BoardForecast While Upstream In Transport Finished State

	ELSE

		fHermesIllegalMsgTransportFiniUS	:= 0;

	END_IF

END_FUNCTION
```

#### fHermesIllegalMsgTransportStopUS.st
```iecst
(* Hermes Illegal Message - Transport Stopped For Upstream *)
FUNCTION fHermesIllegalMsgTransportStopUS

	IF tyMsgType.bServiceDescription = TRUE THEN

		fHermesIllegalMsgTransportStopUS	:= 2833;	//Receive ServiceDescription While Upstream In Transport Stopped State

	ELSIF tyMsgType.bBoardAvailable = TRUE AND bBoardAvailable = TRUE THEN

		fHermesIllegalMsgTransportStopUS	:= 2834;	//Receive Twice Board Available While Upstream In Transport Stopped State

	ELSIF tyMsgType.bRevokeBoardAvailable = TRUE AND bBoardAvailable = FALSE THEN

		fHermesIllegalMsgTransportStopUS	:= 2835;	//Receive RevokeBoardAvailable Without BoardAvailable While Upstream In Transport Stopped State

	ELSIF tyMsgType.bMachineReady = TRUE THEN

		fHermesIllegalMsgTransportStopUS	:= 2836;	//Receive MachineReady While Upstream In Transport Stopped State

	ELSIF tyMsgType.bRevokeMachineReady = TRUE THEN

		fHermesIllegalMsgTransportStopUS	:= 2837;	//Receive RevokeMachineReady While Upstream In Transport Stopped State

	ELSIF tyMsgType.bStartTransport = TRUE THEN

		fHermesIllegalMsgTransportStopUS	:= 2838;	//Receive StartTransport While Upstream In Transport Stopped State

	ELSIF tyMsgType.bStopTransport = TRUE THEN

		fHermesIllegalMsgTransportStopUS	:= 2839;	//Receive StopTransport While Upstream In Transport Stopped State

	ELSE

		fHermesIllegalMsgTransportStopUS	:= 0;

	END_IF

END_FUNCTION
```

#### fHermesIllegalMsgNotConnectedDS.st
```iecst
(* Hermes Illegal Message - Not Connected For Downstream *)
FUNCTION fHermesIllegalMsgNotConnectedDS

	IF tyMsgType.bBoardAvailable = TRUE THEN

		fHermesIllegalMsgNotConnectedDS	:= 2840;	//Receive BoardAvailable While Downstream In Not Connected State

	ELSIF tyMsgType.bRevokeBoardAvailable = TRUE THEN

		fHermesIllegalMsgNotConnectedDS	:= 2841;	//Receive RevokeBoardAvailable While Downstream In Not Connected State

	ELSIF tyMsgType.bMachineReady = TRUE THEN

		fHermesIllegalMsgNotConnectedDS	:= 2842;	//Receive MachineReady While Downstream In Not Connected State

	ELSIF tyMsgType.bRevokeMachineReady = TRUE THEN

		fHermesIllegalMsgNotConnectedDS	:= 2843;	//Receive RevokeMachineReady While Downstream In Not Connected State

	ELSIF tyMsgType.bStartTransport = TRUE THEN

		fHermesIllegalMsgNotConnectedDS	:= 2844;	//Receive StartTransport While Downstream In Not Connected State

	ELSIF tyMsgType.bStopTransport = TRUE THEN

		fHermesIllegalMsgNotConnectedDS	:= 2845;	//Receive StopTransport While Downstream In Not Connected State

	ELSIF tyMsgType.bTransportFinished = TRUE THEN

		fHermesIllegalMsgNotConnectedDS	:= 2846;	//Receive TransportFinished While Downstream In Not Connected State

	ELSIF tyMsgType.bBoardForecast = TRUE THEN

		fHermesIllegalMsgNotConnectedDS	:= 2847;	//Receive BoardForecast While Downstream In Not Connected State

	ELSE

		fHermesIllegalMsgNotConnectedDS	:= 0;

	END_IF

END_FUNCTION
```

#### fHermesIllegalMsgSrvcDescripDS.st
```iecst
(* Hermes Illegal Message - Service Description For Downstream *)
FUNCTION fHermesIllegalMsgSrvcDescripDS

	IF tyMsgType.bServiceDescription = TRUE THEN

		fHermesIllegalMsgSrvcDescripDS	:= 2848;	//Receive ServiceDescription While Downstream In Service Description State

	ELSIF tyMsgType.bBoardAvailable = TRUE THEN

		fHermesIllegalMsgSrvcDescripDS	:= 2849;	//Receive BoardAvailable While Downstream In Service Description State

	ELSIF tyMsgType.bRevokeBoardAvailable = TRUE THEN

		fHermesIllegalMsgSrvcDescripDS	:= 2850;	//Receive RevokeBoardAvailable While Downstream In Service Description State

	ELSIF tyMsgType.bMachineReady = TRUE THEN

		fHermesIllegalMsgSrvcDescripDS	:= 2851;	//Receive MachineReady While Downstream In Service Description State

	ELSIF tyMsgType.bRevokeMachineReady = TRUE THEN

		fHermesIllegalMsgSrvcDescripDS	:= 2852;	//Receive RevokeMachineReady While Downstream In Service Description State

	ELSIF tyMsgType.bStartTransport = TRUE THEN

		fHermesIllegalMsgSrvcDescripDS	:= 2853;	//Receive StartTransport While Downstream In Service Description State

	ELSIF tyMsgType.bStopTransport = TRUE THEN

		fHermesIllegalMsgSrvcDescripDS	:= 2854;	//Receive StopTransport While Downstream In Service Description State

	ELSIF tyMsgType.bTransportFinished = TRUE THEN

		fHermesIllegalMsgSrvcDescripDS	:= 2855;	//Receive TransportFinished While Downstream In Service Description State

	ELSIF tyMsgType.bBoardForecast = TRUE THEN

		fHermesIllegalMsgSrvcDescripDS	:= 2856;	//Receive BoardForecast While Downstream In Service Description State

	ELSE

		fHermesIllegalMsgSrvcDescripDS	:= 0;

	END_IF

END_FUNCTION
```
